LIN {X 0,Y 680.461,Z 406.458,A -85,B 0,C 180,E1 25579.128,E2 25579.128} C_VEL
LIN {X 0,Y 680.451,Z 406.465,A -85,B 0,C 180,E1 25576.563,E2 25576.563} C_VEL
LIN {X 0,Y 680.527,Z 406.447,A -85,B 0,C 180,E1 25573.683,E2 25573.683} C_VEL
LIN {X 0,Y 680.452,Z 406.461,A -85,B 0,C 180,E1 25570.756,E2 25570.756} C_VEL
LIN {X 0,Y 680.448,Z 406.447,A -85,B 0,C 180,E1 25568.195,E2 25568.195} C_VEL
LIN {X 0,Y 680.527,Z 406.46,A -85,B 0,C 180,E1 25565.311,E2 25565.311} C_VEL
LIN {X 0,Y 680.442,Z 406.447,A -85,B 0,C 180,E1 25562.358,E2 25562.358} C_VEL
LIN {X 0,Y 680.451,Z 406.466,A -85,B 0,C 180,E1 25559.832,E2 25559.832} C_VEL
LIN {X 0,Y 680.505,Z 406.442,A -85,B 0,C 180,E1 25556.799,E2 25556.799} C_VEL
LIN {X 0,Y 680.44,Z 406.466,A -85,B 0,C 180,E1 25554.011,E2 25554.011} C_VEL
LIN {X 0,Y 680.446,Z 406.46,A -85,B 0,C 180,E1 25551.55,E2 25551.55} C_VEL
LIN {X 0,Y 680.503,Z 406.464,A -85,B 0,C 180,E1 25548.51,E2 25548.51} C_VEL
LIN {X 0,Y 680.436,Z 406.455,A -85,B 0,C 180,E1 25545.794,E2 25545.794} C_VEL
LIN {X 0,Y 680.437,Z 406.459,A -85,B 0,C 180,E1 25543.338,E2 25543.338} C_VEL
LIN {X 0,Y 680.522,Z 406.444,A -85,B 0,C 180,E1 25540.427,E2 25540.427} C_VEL
LIN {X 0,Y 680.436,Z 406.465,A -85,B 0,C 180,E1 25537.538,E2 25537.538} C_VEL
LIN {X 0,Y 680.434,Z 406.459,A -85,B 0,C 180,E1 25535.038,E2 25535.038} C_VEL
LIN {X 0,Y 680.519,Z 406.463,A -85,B 0,C 180,E1 25532.049,E2 25532.049} C_VEL
LIN {X 0,Y 680.431,Z 406.462,A -85,B 0,C 180,E1 25529.244,E2 25529.244} C_VEL
LIN {X 0,Y 680.43,Z 406.467,A -85,B 0,C 180,E1 25526.762,E2 25526.762} C_VEL
LIN {X 0,Y 680.516,Z 406.467,A -85,B 0,C 180,E1 25523.9,E2 25523.9} C_VEL
LIN {X 0,Y 680.432,Z 406.473,A -85,B 0,C 180,E1 25521.012,E2 25521.012} C_VEL
LIN {X 0,Y 680.426,Z 406.493,A -85,B 0,C 180,E1 25518.714,E2 25518.714} C_VEL
LIN {X 0,Y 681.564,Z 409.672,A -85,B 0,C 180,E1 25518.35,E2 25518.35} C_VEL
LIN {X 0,Y 682.745,Z 411.865,A -85,B 0,C 180,E1 25518.064,E2 25518.064} C_VEL
LIN {X 0,Y 690.51,Z 428.251,A -85,B 0,C 180,E1 25516.112,E2 25516.112} C_VEL
LIN {X 0,Y 698.322,Z 440.196,A -85,B 0,C 180,E1 25515.278,E2 25515.278} C_VEL
LIN {X 0,Y 700.79,Z 450.164,A -85,B 0,C 180,E1 25514.933,E2 25514.933} C_VEL
LIN {X 0,Y 698.561,Z 650.685,A -85,B 0,C 180,E1 25512.321,E2 25512.321} C_VEL
LIN {X 0,Y 696.219,Z 875.891,A -85,B 0,C 180,E1 25509.482,E2 25509.482} C_VEL
LIN {X 0,Y 695.65,Z 912.99,A -85,B 0,C 180,E1 25508.982,E2 25508.982} C_VEL
LIN {X 0,Y 694.867,Z 939.914,A -85,B 0,C 180,E1 25508.45,E2 25508.45} C_VEL
LIN {X 0,Y 694.006,Z 964.483,A -85,B 0,C 180,E1 25507.821,E2 25507.821} C_VEL
LIN {X 0,Y 692.884,Z 992.482,A -85,B 0,C 180,E1 25506.92,E2 25506.92} C_VEL
LIN {X 0,Y 691.785,Z 1015.446,A -85,B 0,C 180,E1 25506.029,E2 25506.029} C_VEL
LIN {X 0,Y 690.755,Z 1035.669,A -85,B 0,C 180,E1 25505.129,E2 25505.129} C_VEL
LIN {X 0,Y 689.672,Z 1055.672,A -85,B 0,C 180,E1 25504.122,E2 25504.122} C_VEL
LIN {X 0,Y 688.5,Z 1076.88,A -85,B 0,C 180,E1 25502.921,E2 25502.921} C_VEL
LIN {X 0,Y 687.043,Z 1101.699,A -85,B 0,C 180,E1 25501.318,E2 25501.318} C_VEL
LIN {X 0,Y 685.98,Z 1120.495,A -85,B 0,C 180,E1 25499.945,E2 25499.945} C_VEL
LIN {X 0,Y 684.979,Z 1138.865,A -85,B 0,C 180,E1 25498.46,E2 25498.46} C_VEL
LIN {X 0,Y 683.778,Z 1160.458,A -85,B 0,C 180,E1 25496.5,E2 25496.5} C_VEL
LIN {X 0,Y 682.976,Z 1176.724,A -85,B 0,C 180,E1 25494.842,E2 25494.842} C_VEL
LIN {X 0,Y 682.182,Z 1193.517,A -85,B 0,C 180,E1 25492.943,E2 25492.943} C_VEL
LIN {X 0,Y 681.485,Z 1209.919,A -85,B 0,C 180,E1 25490.832,E2 25490.832} C_VEL
LIN {X 0,Y 681.039,Z 1222.568,A -85,B 0,C 180,E1 25489.001,E2 25489.001} C_VEL
LIN {X 0,Y 680.648,Z 1234.89,A -85,B 0,C 180,E1 25486.993,E2 25486.993} C_VEL
LIN {X 0,Y 680.344,Z 1246.853,A -85,B 0,C 180,E1 25484.726,E2 25484.726} C_VEL
LIN {X 0,Y 680.165,Z 1255.449,A -85,B 0,C 180,E1 25482.822,E2 25482.822} C_VEL
LIN {X 0,Y 680.027,Z 1262.449,A -85,B 0,C 180,E1 25481.017,E2 25481.017} C_VEL
LIN {X 0,Y 679.932,Z 1268.06,A -85,B 0,C 180,E1 25479.306,E2 25479.306} C_VEL
LIN {X 0,Y 679.922,Z 1273.174,A -85,B 0,C 180,E1 25477.433,E2 25477.433} C_VEL
LIN {X 0,Y 679.916,Z 1277.787,A -85,B 0,C 180,E1 25475.144,E2 25475.144} C_VEL
LIN {X 0,Y 679.912,Z 1280.543,A -85,B 0,C 180,E1 25472.948,E2 25472.948} C_VEL
LIN {X 0,Y 679.88,Z 1281.715,A -85,B 0,C 180,E1 25471.093,E2 25471.093} C_VEL
LIN {X 0,Y 679.863,Z 1281.826,A -85,B 0,C 180,E1 25469.323,E2 25469.323} C_VEL
LIN {X 0,Y 679.906,Z 1280.944,A -85,B 0,C 180,E1 25467.553,E2 25467.553} C_VEL
LIN {X 0,Y 679.915,Z 1278.916,A -85,B 0,C 180,E1 25465.612,E2 25465.612} C_VEL
LIN {X 0,Y 679.929,Z 1274.902,A -85,B 0,C 180,E1 25463.326,E2 25463.326} C_VEL
LIN {X 0,Y 679.942,Z 1269.325,A -85,B 0,C 180,E1 25461.116,E2 25461.116} C_VEL
LIN {X 0,Y 680.018,Z 1263.349,A -85,B 0,C 180,E1 25459.236,E2 25459.236} C_VEL
LIN {X 0,Y 680.138,Z 1256.5,A -85,B 0,C 180,E1 25457.431,E2 25457.431} C_VEL
LIN {X 0,Y 680.313,Z 1248.061,A -85,B 0,C 180,E1 25455.529,E2 25455.529} C_VEL
LIN {X 0,Y 680.558,Z 1237.337,A -85,B 0,C 180,E1 25453.438,E2 25453.438} C_VEL
LIN {X 0,Y 681.006,Z 1223.582,A -85,B 0,C 180,E1 25451.153,E2 25451.153} C_VEL
LIN {X 0,Y 681.419,Z 1211.446,A -85,B 0,C 180,E1 25449.379,E2 25449.379} C_VEL
LIN {X 0,Y 681.994,Z 1197.829,A -85,B 0,C 180,E1 25447.591,E2 25447.591} C_VEL
LIN {X 0,Y 682.821,Z 1180.065,A -85,B 0,C 180,E1 25445.516,E2 25445.516} C_VEL
LIN {X 0,Y 683.651,Z 1163.367,A -85,B 0,C 180,E1 25443.786,E2 25443.786} C_VEL
LIN {X 0,Y 684.531,Z 1146.227,A -85,B 0,C 180,E1 25442.179,E2 25442.179} C_VEL
LIN {X 0,Y 685.783,Z 1124.207,A -85,B 0,C 180,E1 25440.341,E2 25440.341} C_VEL
LIN {X 0,Y 686.866,Z 1105.212,A -85,B 0,C 180,E1 25438.931,E2 25438.931} C_VEL
LIN {X 0,Y 687.971,Z 1085.491,A -85,B 0,C 180,E1 25437.61,E2 25437.61} C_VEL
LIN {X 0,Y 689.442,Z 1059.964,A -85,B 0,C 180,E1 25436.107,E2 25436.107} C_VEL
LIN {X 0,Y 690.596,Z 1038.67,A -85,B 0,C 180,E1 25435.015,E2 25435.015} C_VEL
LIN {X 0,Y 691.623,Z 1018.703,A -85,B 0,C 180,E1 25434.109,E2 25434.109} C_VEL
LIN {X 0,Y 692.595,Z 998.275,A -85,B 0,C 180,E1 25433.295,E2 25433.295} C_VEL
LIN {X 0,Y 693.53,Z 975.906,A -85,B 0,C 180,E1 25432.524,E2 25432.524} C_VEL
LIN {X 0,Y 694.564,Z 949.817,A -85,B 0,C 180,E1 25431.784,E2 25431.784} C_VEL
LIN {X 0,Y 695.356,Z 923.501,A -85,B 0,C 180,E1 25431.208,E2 25431.208} C_VEL
LIN {X 0,Y 695.924,Z 898.793,A -85,B 0,C 180,E1 25430.808,E2 25430.808} C_VEL
LIN {X 0,Y 698.307,Z 673.627,A -85,B 0,C 180,E1 25427.971,E2 25427.971} C_VEL
LIN {X 0,Y 700.497,Z 475.392,A -85,B 0,C 180,E1 25425.4,E2 25425.4} C_VEL
LIN {X 0,Y 700.649,Z 448.932,A -85,B 0,C 180,E1 25425.038,E2 25425.038} C_VEL
LIN {X 0,Y 697.841,Z 439.159,A -85,B 0,C 180,E1 25424.667,E2 25424.667} C_VEL
LIN {X 0,Y 690.054,Z 427.342,A -85,B 0,C 180,E1 25423.812,E2 25423.812} C_VEL
LIN {X 0,Y 683.62,Z 413.795,A -85,B 0,C 180,E1 25422.172,E2 25422.172} C_VEL
LIN {X 0,Y 681.91,Z 410.194,A -85,B 0,C 180,E1 25421.724,E2 25421.724} C_VEL
LIN {X 0,Y 680.512,Z 407.036,A -85,B 0,C 180,E1 25421.338,E2 25421.338} C_VEL
LIN {X 0,Y 680.421,Z 406.454,A -85,B 0,C 180,E1 25421.258,E2 25421.258} C_VEL
LIN {X 0,Y 680.51,Z 406.449,A -85,B 0,C 180,E1 25418.428,E2 25418.428} C_VEL
LIN {X 0,Y 680.436,Z 406.469,A -85,B 0,C 180,E1 25415.482,E2 25415.482} C_VEL
LIN {X 0,Y 680.436,Z 406.462,A -85,B 0,C 180,E1 25413.037,E2 25413.037} C_VEL
LIN {X 0,Y 680.529,Z 406.444,A -85,B 0,C 180,E1 25410.165,E2 25410.165} C_VEL
LIN {X 0,Y 680.45,Z 406.466,A -85,B 0,C 180,E1 25407.25,E2 25407.25} C_VEL
LIN {X 0,Y 680.457,Z 406.449,A -85,B 0,C 180,E1 25404.666,E2 25404.666} C_VEL
LIN {X 0,Y 680.512,Z 406.452,A -85,B 0,C 180,E1 25401.642,E2 25401.642} C_VEL
LIN {X 0,Y 680.456,Z 406.459,A -85,B 0,C 180,E1 25398.859,E2 25398.859} C_VEL
LIN {X 0,Y 680.513,Z 406.451,A -85,B 0,C 180,E1 25396.036,E2 25396.036} C_VEL
LIN {X 0,Y 680.476,Z 406.46,A -85,B 0,C 180,E1 25392.992,E2 25392.992} C_VEL
LIN {X 0,Y 680.483,Z 406.459,A -85,B 0,C 180,E1 25390.241,E2 25390.241} C_VEL
LIN {X 0,Y 680.508,Z 406.458,A -85,B 0,C 180,E1 25387.09,E2 25387.09} C_VEL
LIN {X 0,Y 680.483,Z 406.459,A -85,B 0,C 180,E1 25384.213,E2 25384.213} C_VEL
LIN {X 0,Y 680.525,Z 406.457,A -85,B 0,C 180,E1 25381.179,E2 25381.179} C_VEL
LIN {X 0,Y 680.485,Z 406.459,A -85,B 0,C 180,E1 25378.232,E2 25378.232} C_VEL
LIN {X 0,Y 680.518,Z 406.46,A -85,B 0,C 180,E1 25375.28,E2 25375.28} C_VEL
LIN {X 0,Y 680.494,Z 406.456,A -85,B 0,C 180,E1 25372.316,E2 25372.316} C_VEL
LIN {X 0,Y 680.517,Z 406.456,A -85,B 0,C 180,E1 25369.331,E2 25369.331} C_VEL
LIN {X 0,Y 680.509,Z 406.452,A -85,B 0,C 180,E1 25366.316,E2 25366.316} C_VEL
LIN {X 0,Y 680.519,Z 406.46,A -85,B 0,C 180,E1 25363.263,E2 25363.263} C_VEL
LIN {X 0,Y 680.515,Z 406.446,A -85,B 0,C 180,E1 25360.159,E2 25360.159} C_VEL
LIN {X 0,Y 680.513,Z 406.465,A -85,B 0,C 180,E1 25357.085,E2 25357.085} C_VEL
LIN {X 0,Y 680.52,Z 406.44,A -85,B 0,C 180,E1 25354.033,E2 25354.033} C_VEL
LIN {X 0,Y 680.509,Z 406.452,A -85,B 0,C 180,E1 25350.956,E2 25350.956} C_VEL
LIN {X 0,Y 680.514,Z 406.444,A -85,B 0,C 180,E1 25349.429,E2 25349.429} C_VEL
LIN {X 0,Y 679.535,Z 406.579,A -85,B 0,C 180,E1 25348.78,E2 25348.78} C_VEL
LIN {X 0,Y 673.085,Z 407.384,A -85,B 0,C 180,E1 25346.963,E2 25346.963} C_VEL
LIN {X 0,Y 672.552,Z 407.44,A -85,B 0,C 180,E1 25346.49,E2 25346.49} C_VEL
LIN {X 0,Y 672.581,Z 407.453,A -85,B 0,C 180,E1 25343.511,E2 25343.511} C_VEL
LIN {X 0,Y 672.548,Z 407.456,A -85,B 0,C 180,E1 25340.482,E2 25340.482} C_VEL
LIN {X 0,Y 672.577,Z 407.645,A -85,B 0,C 180,E1 25338.551,E2 25338.551} C_VEL
LIN {X 0,Y 673.992,Z 411.125,A -85,B 0,C 180,E1 25338.118,E2 25338.118} C_VEL
LIN {X 0,Y 677.306,Z 418.165,A -85,B 0,C 180,E1 25337.242,E2 25337.242} C_VEL
LIN {X 0,Y 690.16,Z 436.862,A -85,B 0,C 180,E1 25335.824,E2 25335.824} C_VEL
LIN {X 0,Y 695.097,Z 444.613,A -85,B 0,C 180,E1 25335.294,E2 25335.294} C_VEL
LIN {X 0,Y 692.495,Z 652.368,A -85,B 0,C 180,E1 25332.574,E2 25332.574} C_VEL
LIN {X 0,Y 689.915,Z 876.906,A -85,B 0,C 180,E1 25329.723,E2 25329.723} C_VEL
LIN {X 0,Y 689.283,Z 907.492,A -85,B 0,C 180,E1 25329.277,E2 25329.277} C_VEL
LIN {X 0,Y 688.468,Z 932.192,A -85,B 0,C 180,E1 25328.77,E2 25328.77} C_VEL
LIN {X 0,Y 687.491,Z 957.703,A -85,B 0,C 180,E1 25328.098,E2 25328.098} C_VEL
LIN {X 0,Y 686.246,Z 984.6,A -85,B 0,C 180,E1 25327.206,E2 25327.206} C_VEL
LIN {X 0,Y 685.151,Z 1005.466,A -85,B 0,C 180,E1 25326.388,E2 25326.388} C_VEL
LIN {X 0,Y 684.005,Z 1025.807,A -85,B 0,C 180,E1 25325.475,E2 25325.475} C_VEL
LIN {X 0,Y 682.824,Z 1045.645,A -85,B 0,C 180,E1 25324.469,E2 25324.469} C_VEL
LIN {X 0,Y 681.518,Z 1066.981,A -85,B 0,C 180,E1 25323.251,E2 25323.251} C_VEL
LIN {X 0,Y 679.929,Z 1091.276,A -85,B 0,C 180,E1 25321.669,E2 25321.669} C_VEL
LIN {X 0,Y 678.72,Z 1110.473,A -85,B 0,C 180,E1 25320.255,E2 25320.255} C_VEL
LIN {X 0,Y 677.602,Z 1128.839,A -85,B 0,C 180,E1 25318.756,E2 25318.756} C_VEL
LIN {X 0,Y 676.295,Z 1150.13,A -85,B 0,C 180,E1 25316.805,E2 25316.805} C_VEL
LIN {X 0,Y 675.369,Z 1166.266,A -85,B 0,C 180,E1 25315.146,E2 25315.146} C_VEL
LIN {X 0,Y 674.542,Z 1182.325,A -85,B 0,C 180,E1 25313.316,E2 25313.316} C_VEL
LIN {X 0,Y 673.736,Z 1199.196,A -85,B 0,C 180,E1 25311.141,E2 25311.141} C_VEL
LIN {X 0,Y 673.208,Z 1212.129,A -85,B 0,C 180,E1 25309.254,E2 25309.254} C_VEL
LIN {X 0,Y 672.776,Z 1223.563,A -85,B 0,C 180,E1 25307.383,E2 25307.383} C_VEL
LIN {X 0,Y 672.406,Z 1236.211,A -85,B 0,C 180,E1 25304.997,E2 25304.997} C_VEL
LIN {X 0,Y 672.191,Z 1245.602,A -85,B 0,C 180,E1 25302.895,E2 25302.895} C_VEL
LIN {X 0,Y 672.049,Z 1252.579,A -85,B 0,C 180,E1 25301.067,E2 25301.067} C_VEL
LIN {X 0,Y 671.94,Z 1258.169,A -85,B 0,C 180,E1 25299.337,E2 25299.337} C_VEL
LIN {X 0,Y 671.92,Z 1263.258,A -85,B 0,C 180,E1 25297.441,E2 25297.441} C_VEL
LIN {X 0,Y 671.916,Z 1267.7,A -85,B 0,C 180,E1 25295.21,E2 25295.21} C_VEL
LIN {X 0,Y 671.911,Z 1270.503,A -85,B 0,C 180,E1 25292.988,E2 25292.988} C_VEL
LIN {X 0,Y 671.88,Z 1271.725,A -85,B 0,C 180,E1 25291.026,E2 25291.026} C_VEL
LIN {X 0,Y 671.863,Z 1271.817,A -85,B 0,C 180,E1 25289.235,E2 25289.235} C_VEL
LIN {X 0,Y 671.904,Z 1270.917,A -85,B 0,C 180,E1 25287.444,E2 25287.444} C_VEL
LIN {X 0,Y 671.911,Z 1268.866,A -85,B 0,C 180,E1 25285.479,E2 25285.479} C_VEL
LIN {X 0,Y 671.928,Z 1264.831,A -85,B 0,C 180,E1 25283.166,E2 25283.166} C_VEL
LIN {X 0,Y 671.944,Z 1259.472,A -85,B 0,C 180,E1 25281.014,E2 25281.014} C_VEL
LIN {X 0,Y 672.028,Z 1253.526,A -85,B 0,C 180,E1 25279.111,E2 25279.111} C_VEL
LIN {X 0,Y 672.179,Z 1246.349,A -85,B 0,C 180,E1 25277.198,E2 25277.198} C_VEL
LIN {X 0,Y 672.363,Z 1238.295,A -85,B 0,C 180,E1 25275.359,E2 25275.359} C_VEL
LIN {X 0,Y 672.626,Z 1228.064,A -85,B 0,C 180,E1 25273.331,E2 25273.331} C_VEL
LIN {X 0,Y 673.118,Z 1214.475,A -85,B 0,C 180,E1 25271.019,E2 25271.019} C_VEL
LIN {X 0,Y 673.606,Z 1201.803,A -85,B 0,C 180,E1 25269.134,E2 25269.134} C_VEL
LIN {X 0,Y 674.234,Z 1188.219,A -85,B 0,C 180,E1 25267.324,E2 25267.324} C_VEL
LIN {X 0,Y 675.186,Z 1170.313,A -85,B 0,C 180,E1 25265.204,E2 25265.204} C_VEL
LIN {X 0,Y 676.1,Z 1153.397,A -85,B 0,C 180,E1 25263.429,E2 25263.429} C_VEL
LIN {X 0,Y 677.123,Z 1136.253,A -85,B 0,C 180,E1 25261.805,E2 25261.805} C_VEL
LIN {X 0,Y 678.509,Z 1114.078,A -85,B 0,C 180,E1 25259.935,E2 25259.935} C_VEL
LIN {X 0,Y 679.729,Z 1094.572,A -85,B 0,C 180,E1 25258.475,E2 25258.475} C_VEL
LIN {X 0,Y 681.026,Z 1074.12,A -85,B 0,C 180,E1 25257.1,E2 25257.1} C_VEL
LIN {X 0,Y 682.626,Z 1049.079,A -85,B 0,C 180,E1 25255.626,E2 25255.626} C_VEL
LIN {X 0,Y 683.902,Z 1027.662,A -85,B 0,C 180,E1 25254.524,E2 25254.524} C_VEL
LIN {X 0,Y 685.039,Z 1007.552,A -85,B 0,C 180,E1 25253.611,E2 25253.611} C_VEL
LIN {X 0,Y 686.085,Z 987.66,A -85,B 0,C 180,E1 25252.818,E2 25252.818} C_VEL
LIN {X 0,Y 687.13,Z 965.185,A -85,B 0,C 180,E1 25252.043,E2 25252.043} C_VEL
LIN {X 0,Y 688.273,Z 938.268,A -85,B 0,C 180,E1 25251.284,E2 25251.284} C_VEL
LIN {X 0,Y 689.108,Z 912.632,A -85,B 0,C 180,E1 25250.727,E2 25250.727} C_VEL
LIN {X 0,Y 689.74,Z 887.818,A -85,B 0,C 180,E1 25250.328,E2 25250.328} C_VEL
LIN {X 0,Y 692.374,Z 662.26,A -85,B 0,C 180,E1 25247.464,E2 25247.464} C_VEL
LIN {X 0,Y 694.923,Z 457.036,A -85,B 0,C 180,E1 25244.78,E2 25244.78} C_VEL
LIN {X 0,Y 694.963,Z 444.111,A -85,B 0,C 180,E1 25244.597,E2 25244.597} C_VEL
LIN {X 0,Y 681.325,Z 423.894,A -85,B 0,C 180,E1 25243.12,E2 25243.12} C_VEL
LIN {X 0,Y 677.021,Z 417.66,A -85,B 0,C 180,E1 25242.622,E2 25242.622} C_VEL
LIN {X 0,Y 673.899,Z 411.027,A -85,B 0,C 180,E1 25241.775,E2 25241.775} C_VEL
LIN {X 0,Y 672.527,Z 407.436,A -85,B 0,C 180,E1 25241.31,E2 25241.31} C_VEL
LIN {X 0,Y 672.583,Z 407.454,A -85,B 0,C 180,E1 25238.292,E2 25238.292} C_VEL
LIN {X 0,Y 672.52,Z 407.454,A -85,B 0,C 180,E1 25235.44,E2 25235.44} C_VEL
LIN {X 0,Y 672.559,Z 407.45,A -85,B 0,C 180,E1 25232.661,E2 25232.661} C_VEL
LIN {X 0,Y 672.533,Z 407.44,A -85,B 0,C 180,E1 25229.578,E2 25229.578} C_VEL
LIN {X 0,Y 672.517,Z 407.454,A -85,B 0,C 180,E1 25226.967,E2 25226.967} C_VEL
LIN {X 0,Y 672.588,Z 407.442,A -85,B 0,C 180,E1 25224.038,E2 25224.038} C_VEL
LIN {X 0,Y 672.516,Z 407.442,A -85,B 0,C 180,E1 25221.088,E2 25221.088} C_VEL
LIN {X 0,Y 672.522,Z 407.449,A -85,B 0,C 180,E1 25218.463,E2 25218.463} C_VEL
LIN {X 0,Y 672.569,Z 407.427,A -85,B 0,C 180,E1 25215.433,E2 25215.433} C_VEL
LIN {X 0,Y 672.508,Z 407.452,A -85,B 0,C 180,E1 25212.625,E2 25212.625} C_VEL
LIN {X 0,Y 672.538,Z 407.443,A -85,B 0,C 180,E1 25209.931,E2 25209.931} C_VEL
LIN {X 0,Y 672.529,Z 407.452,A -85,B 0,C 180,E1 25206.831,E2 25206.831} C_VEL
LIN {X 0,Y 672.503,Z 407.449,A -85,B 0,C 180,E1 25204.263,E2 25204.263} C_VEL
LIN {X 0,Y 672.56,Z 407.438,A -85,B 0,C 180,E1 25201.448,E2 25201.448} C_VEL
LIN {X 0,Y 672.518,Z 407.447,A -85,B 0,C 180,E1 25198.466,E2 25198.466} C_VEL
LIN {X 0,Y 672.5,Z 407.438,A -85,B 0,C 180,E1 25195.907,E2 25195.907} C_VEL
LIN {X 0,Y 672.57,Z 407.454,A -85,B 0,C 180,E1 25193.084,E2 25193.084} C_VEL
LIN {X 0,Y 672.506,Z 407.44,A -85,B 0,C 180,E1 25190.068,E2 25190.068} C_VEL
LIN {X 0,Y 672.499,Z 407.456,A -85,B 0,C 180,E1 25187.55,E2 25187.55} C_VEL
LIN {X 0,Y 672.583,Z 407.429,A -85,B 0,C 180,E1 25184.655,E2 25184.655} C_VEL
LIN {X 0,Y 672.501,Z 407.453,A -85,B 0,C 180,E1 25181.716,E2 25181.716} C_VEL
LIN {X 0,Y 672.495,Z 407.432,A -85,B 0,C 180,E1 25179.185,E2 25179.185} C_VEL
LIN {X 0,Y 672.582,Z 407.446,A -85,B 0,C 180,E1 25176.241,E2 25176.241} C_VEL
LIN {X 0,Y 672.492,Z 407.452,A -85,B 0,C 180,E1 25173.317,E2 25173.317} C_VEL
LIN {X 0,Y 672.493,Z 407.454,A -85,B 0,C 180,E1 25170.909,E2 25170.909} C_VEL
LIN {X 0,Y 672.58,Z 407.454,A -85,B 0,C 180,E1 25168.045,E2 25168.045} C_VEL
LIN {X 0,Y 672.49,Z 407.45,A -85,B 0,C 180,E1 25165.079,E2 25165.079} C_VEL
LIN {X 0,Y 672.493,Z 407.459,A -85,B 0,C 180,E1 25162.551,E2 25162.551} C_VEL
LIN {X 0,Y 672.563,Z 407.436,A -85,B 0,C 180,E1 25159.561,E2 25159.561} C_VEL
LIN {X 0,Y 672.57,Z 407.709,A -85,B 0,C 180,E1 25159.371,E2 25159.371} C_VEL
LIN {X 0,Y 673.708,Z 410.787,A -85,B 0,C 180,E1 25159.004,E2 25159.004} C_VEL
LIN {X 0,Y 674.92,Z 413.31,A -85,B 0,C 180,E1 25158.68,E2 25158.68} C_VEL
LIN {X 0,Y 679.079,Z 421.931,A -85,B 0,C 180,E1 25157.595,E2 25157.595} C_VEL
LIN {X 0,Y 682.242,Z 428.302,A -85,B 0,C 180,E1 25156.838,E2 25156.838} C_VEL
LIN {X 0,Y 693.373,Z 445.15,A -85,B 0,C 180,E1 25155.621,E2 25155.621} C_VEL
LIN {X 0,Y 695.087,Z 452.546,A -85,B 0,C 180,E1 25155.37,E2 25155.37} C_VEL
LIN {X 0,Y 692.614,Z 652.848,A -85,B 0,C 180,E1 25152.741,E2 25152.741} C_VEL
LIN {X 0,Y 690.015,Z 878.054,A -85,B 0,C 180,E1 25149.879,E2 25149.879} C_VEL
LIN {X 0,Y 689.393,Z 913.685,A -85,B 0,C 180,E1 25149.39,E2 25149.39} C_VEL
LIN {X 0,Y 688.544,Z 940.238,A -85,B 0,C 180,E1 25148.86,E2 25148.86} C_VEL
LIN {X 0,Y 687.611,Z 964.53,A -85,B 0,C 180,E1 25148.234,E2 25148.234} C_VEL
LIN {X 0,Y 686.378,Z 992.125,A -85,B 0,C 180,E1 25147.344,E2 25147.344} C_VEL
LIN {X 0,Y 685.15,Z 1015.443,A -85,B 0,C 180,E1 25146.434,E2 25146.434} C_VEL
LIN {X 0,Y 684.005,Z 1035.795,A -85,B 0,C 180,E1 25145.521,E2 25145.521} C_VEL
LIN {X 0,Y 682.826,Z 1055.62,A -85,B 0,C 180,E1 25144.516,E2 25144.516} C_VEL
LIN {X 0,Y 681.499,Z 1077.329,A -85,B 0,C 180,E1 25143.275,E2 25143.275} C_VEL
LIN {X 0,Y 679.882,Z 1101.964,A -85,B 0,C 180,E1 25141.666,E2 25141.666} C_VEL
LIN {X 0,Y 678.728,Z 1120.322,A -85,B 0,C 180,E1 25140.312,E2 25140.312} C_VEL
LIN {X 0,Y 677.629,Z 1138.312,A -85,B 0,C 180,E1 25138.845,E2 25138.845} C_VEL
LIN {X 0,Y 676.291,Z 1160.16,A -85,B 0,C 180,E1 25136.847,E2 25136.847} C_VEL
LIN {X 0,Y 675.386,Z 1175.872,A -85,B 0,C 180,E1 25135.234,E2 25135.234} C_VEL
LIN {X 0,Y 674.604,Z 1191.204,A -85,B 0,C 180,E1 25133.494,E2 25133.494} C_VEL
LIN {X 0,Y 673.76,Z 1208.71,A -85,B 0,C 180,E1 25131.254,E2 25131.254} C_VEL
LIN {X 0,Y 673.218,Z 1221.869,A -85,B 0,C 180,E1 25129.339,E2 25129.339} C_VEL
LIN {X 0,Y 672.774,Z 1233.63,A -85,B 0,C 180,E1 25127.416,E2 25127.416} C_VEL
LIN {X 0,Y 672.399,Z 1246.444,A -85,B 0,C 180,E1 25124.992,E2 25124.992} C_VEL
LIN {X 0,Y 672.192,Z 1255.45,A -85,B 0,C 180,E1 25122.977,E2 25122.977} C_VEL
LIN {X 0,Y 672.05,Z 1262.45,A -85,B 0,C 180,E1 25121.149,E2 25121.149} C_VEL
LIN {X 0,Y 671.943,Z 1268.061,A -85,B 0,C 180,E1 25119.418,E2 25119.418} C_VEL
LIN {X 0,Y 671.923,Z 1273.171,A -85,B 0,C 180,E1 25117.522,E2 25117.522} C_VEL
LIN {X 0,Y 671.916,Z 1277.639,A -85,B 0,C 180,E1 25115.291,E2 25115.291} C_VEL
LIN {X 0,Y 671.91,Z 1280.475,A -85,B 0,C 180,E1 25113.068,E2 25113.068} C_VEL
LIN {X 0,Y 671.881,Z 1281.715,A -85,B 0,C 180,E1 25111.106,E2 25111.106} C_VEL
LIN {X 0,Y 671.863,Z 1281.826,A -85,B 0,C 180,E1 25109.315,E2 25109.315} C_VEL
LIN {X 0,Y 671.906,Z 1280.945,A -85,B 0,C 180,E1 25107.524,E2 25107.524} C_VEL
LIN {X 0,Y 671.913,Z 1278.913,A -85,B 0,C 180,E1 25105.56,E2 25105.56} C_VEL
LIN {X 0,Y 671.929,Z 1274.902,A -85,B 0,C 180,E1 25103.247,E2 25103.247} C_VEL
LIN {X 0,Y 671.947,Z 1269.579,A -85,B 0,C 180,E1 25101.095,E2 25101.095} C_VEL
LIN {X 0,Y 672.033,Z 1263.349,A -85,B 0,C 180,E1 25099.106,E2 25099.106} C_VEL
LIN {X 0,Y 672.176,Z 1256.501,A -85,B 0,C 180,E1 25097.28,E2 25097.28} C_VEL
LIN {X 0,Y 672.368,Z 1248.063,A -85,B 0,C 180,E1 25095.354,E2 25095.354} C_VEL
LIN {X 0,Y 672.673,Z 1236.873,A -85,B 0,C 180,E1 25093.149,E2 25093.149} C_VEL
LIN {X 0,Y 673.152,Z 1223.583,A -85,B 0,C 180,E1 25090.925,E2 25090.925} C_VEL
LIN {X 0,Y 673.655,Z 1210.803,A -85,B 0,C 180,E1 25089.039,E2 25089.039} C_VEL
LIN {X 0,Y 674.369,Z 1195.629,A -85,B 0,C 180,E1 25087.038,E2 25087.038} C_VEL
LIN {X 0,Y 675.304,Z 1177.848,A -85,B 0,C 180,E1 25084.98,E2 25084.98} C_VEL
LIN {X 0,Y 676.176,Z 1161.97,A -85,B 0,C 180,E1 25083.332,E2 25083.332} C_VEL
LIN {X 0,Y 677.398,Z 1142.666,A -85,B 0,C 180,E1 25081.524,E2 25081.524} C_VEL
LIN {X 0,Y 678.615,Z 1122.24,A -85,B 0,C 180,E1 25079.837,E2 25079.837} C_VEL
LIN {X 0,Y 679.764,Z 1103.887,A -85,B 0,C 180,E1 25078.471,E2 25078.471} C_VEL
LIN {X 0,Y 681.2,Z 1081.901,A -85,B 0,C 180,E1 25077.004,E2 25077.004} C_VEL
LIN {X 0,Y 682.727,Z 1057.297,A -85,B 0,C 180,E1 25075.575,E2 25075.575} C_VEL
LIN {X 0,Y 683.959,Z 1036.686,A -85,B 0,C 180,E1 25074.522,E2 25074.522} C_VEL
LIN {X 0,Y 685.099,Z 1016.445,A -85,B 0,C 180,E1 25073.609,E2 25073.609} C_VEL
LIN {X 0,Y 686.227,Z 994.996,A -85,B 0,C 180,E1 25072.764,E2 25072.764} C_VEL
LIN {X 0,Y 687.509,Z 967.115,A -85,B 0,C 180,E1 25071.839,E2 25071.839} C_VEL
LIN {X 0,Y 688.482,Z 941.865,A -85,B 0,C 180,E1 25071.177,E2 25071.177} C_VEL
LIN {X 0,Y 689.299,Z 916.908,A -85,B 0,C 180,E1 25070.667,E2 25070.667} C_VEL
LIN {X 0,Y 689.938,Z 884.658,A -85,B 0,C 180,E1 25070.203,E2 25070.203} C_VEL
LIN {X 0,Y 692.523,Z 660.013,A -85,B 0,C 180,E1 25067.351,E2 25067.351} C_VEL
LIN {X 0,Y 694.974,Z 461.158,A -85,B 0,C 180,E1 25064.745,E2 25064.745} C_VEL
LIN {X 0,Y 694.945,Z 451.203,A -85,B 0,C 180,E1 25064.599,E2 25064.599} C_VEL
LIN {X 0,Y 692.933,Z 444.186,A -85,B 0,C 180,E1 25064.328,E2 25064.328} C_VEL
LIN {X 0,Y 681.791,Z 427.694,A -85,B 0,C 180,E1 25063.112,E2 25063.112} C_VEL
LIN {X 0,Y 676.078,Z 415.52,A -85,B 0,C 180,E1 25061.61,E2 25061.61} C_VEL
LIN {X 0,Y 673.709,Z 410.783,A -85,B 0,C 180,E1 25060.996,E2 25060.996} C_VEL
LIN {X 0,Y 672.548,Z 407.436,A -85,B 0,C 180,E1 25060.596,E2 25060.596} C_VEL
LIN {X 0,Y 672.495,Z 407.442,A -85,B 0,C 180,E1 25057.581,E2 25057.581} C_VEL
LIN {X 0,Y 672.494,Z 407.456,A -85,B 0,C 180,E1 25055.128,E2 25055.128} C_VEL
LIN {X 0,Y 672.566,Z 407.452,A -85,B 0,C 180,E1 25052.358,E2 25052.358} C_VEL
LIN {X 0,Y 672.51,Z 407.444,A -85,B 0,C 180,E1 25049.383,E2 25049.383} C_VEL
LIN {X 0,Y 672.51,Z 407.457,A -85,B 0,C 180,E1 25046.864,E2 25046.864} C_VEL
LIN {X 0,Y 672.588,Z 407.446,A -85,B 0,C 180,E1 25043.851,E2 25043.851} C_VEL
LIN {X 0,Y 672.515,Z 407.443,A -85,B 0,C 180,E1 25040.981,E2 25040.981} C_VEL
LIN {X 0,Y 672.56,Z 407.451,A -85,B 0,C 180,E1 25038.192,E2 25038.192} C_VEL
LIN {X 0,Y 672.533,Z 407.429,A -85,B 0,C 180,E1 25035.081,E2 25035.081} C_VEL
LIN {X 0,Y 672.537,Z 407.453,A -85,B 0,C 180,E1 25032.362,E2 25032.362} C_VEL
LIN {X 0,Y 672.574,Z 407.424,A -85,B 0,C 180,E1 25029.239,E2 25029.239} C_VEL
LIN {X 0,Y 672.539,Z 407.452,A -85,B 0,C 180,E1 25026.316,E2 25026.316} C_VEL
LIN {X 0,Y 672.582,Z 407.424,A -85,B 0,C 180,E1 25023.324,E2 25023.324} C_VEL
LIN {X 0,Y 672.545,Z 407.45,A -85,B 0,C 180,E1 25020.341,E2 25020.341} C_VEL
LIN {X 0,Y 672.579,Z 407.427,A -85,B 0,C 180,E1 25017.444,E2 25017.444} C_VEL
LIN {X 0,Y 672.553,Z 407.448,A -85,B 0,C 180,E1 25014.369,E2 25014.369} C_VEL
LIN {X 0,Y 672.582,Z 407.429,A -85,B 0,C 180,E1 25011.45,E2 25011.45} C_VEL
LIN {X 0,Y 672.568,Z 407.447,A -85,B 0,C 180,E1 25008.335,E2 25008.335} C_VEL
LIN {X 0,Y 672.577,Z 407.429,A -85,B 0,C 180,E1 25005.273,E2 25005.273} C_VEL
LIN {X 0,Y 672.573,Z 407.448,A -85,B 0,C 180,E1 25002.166,E2 25002.166} C_VEL
LIN {X 0,Y 672.572,Z 407.434,A -85,B 0,C 180,E1 24999.096,E2 24999.096} C_VEL
LIN {X 0,Y 672.581,Z 407.445,A -85,B 0,C 180,E1 24996.055,E2 24996.055} C_VEL
LIN {X 0,Y 672.568,Z 407.45,A -85,B 0,C 180,E1 24992.938,E2 24992.938} C_VEL
LIN {X 0,Y 672.586,Z 407.428,A -85,B 0,C 180,E1 24989.908,E2 24989.908} C_VEL
LIN {X 0,Y 672.563,Z 407.444,A -85,B 0,C 180,E1 24986.825,E2 24986.825} C_VEL
LIN {X 0,Y 672.552,Z 407.44,A -85,B 0,C 180,E1 24986.49,E2 24986.49} C_VEL
LIN {X 0,Y 671.572,Z 407.559,A -85,B 0,C 180,E1 24985.834,E2 24985.834} C_VEL
LIN {X 0,Y 665.177,Z 408.374,A -85,B 0,C 180,E1 24983.995,E2 24983.995} C_VEL
LIN {X 0,Y 664.642,Z 408.442,A -85,B 0,C 180,E1 24983.517,E2 24983.517} C_VEL
LIN {X 0,Y 664.609,Z 408.443,A -85,B 0,C 180,E1 24980.476,E2 24980.476} C_VEL
LIN {X 0,Y 664.645,Z 408.443,A -85,B 0,C 180,E1 24979.273,E2 24979.273} C_VEL
LIN {X 0,Y 665.818,Z 411.714,A -85,B 0,C 180,E1 24978.87,E2 24978.87} C_VEL
LIN {X 0,Y 666.949,Z 414.048,A -85,B 0,C 180,E1 24978.556,E2 24978.556} C_VEL
LIN {X 0,Y 669.13,Z 418.392,A -85,B 0,C 180,E1 24978.004,E2 24978.004} C_VEL
LIN {X 0,Y 684.846,Z 441.054,A -85,B 0,C 180,E1 24976.222,E2 24976.222} C_VEL
LIN {X 0,Y 689.41,Z 448.321,A -85,B 0,C 180,E1 24975.72,E2 24975.72} C_VEL
LIN {X 0,Y 686.562,Z 655.4,A -85,B 0,C 180,E1 24972.988,E2 24972.988} C_VEL
LIN {X 0,Y 683.716,Z 880.638,A -85,B 0,C 180,E1 24970.107,E2 24970.107} C_VEL
LIN {X 0,Y 683.026,Z 908.798,A -85,B 0,C 180,E1 24969.68,E2 24969.68} C_VEL
LIN {X 0,Y 682.165,Z 932.85,A -85,B 0,C 180,E1 24969.18,E2 24969.18} C_VEL
LIN {X 0,Y 681.071,Z 958.778,A -85,B 0,C 180,E1 24968.488,E2 24968.488} C_VEL
LIN {X 0,Y 679.712,Z 985.319,A -85,B 0,C 180,E1 24967.596,E2 24967.596} C_VEL
LIN {X 0,Y 678.487,Z 1006.607,A -85,B 0,C 180,E1 24966.751,E2 24966.751} C_VEL
LIN {X 0,Y 677.219,Z 1027.124,A -85,B 0,C 180,E1 24965.818,E2 24965.818} C_VEL
LIN {X 0,Y 675.839,Z 1048.303,A -85,B 0,C 180,E1 24964.723,E2 24964.723} C_VEL
LIN {X 0,Y 674.166,Z 1072.717,A -85,B 0,C 180,E1 24963.283,E2 24963.283} C_VEL
LIN {X 0,Y 672.632,Z 1093.952,A -85,B 0,C 180,E1 24961.853,E2 24961.853} C_VEL
LIN {X 0,Y 671.319,Z 1113.05,A -85,B 0,C 180,E1 24960.414,E2 24960.414} C_VEL
LIN {X 0,Y 669.823,Z 1135.25,A -85,B 0,C 180,E1 24958.536,E2 24958.536} C_VEL
LIN {X 0,Y 668.616,Z 1152.932,A -85,B 0,C 180,E1 24956.85,E2 24956.85} C_VEL
LIN {X 0,Y 667.64,Z 1168.815,A -85,B 0,C 180,E1 24955.173,E2 24955.173} C_VEL
LIN {X 0,Y 666.595,Z 1186.78,A -85,B 0,C 180,E1 24953.049,E2 24953.049} C_VEL
LIN {X 0,Y 665.859,Z 1201.136,A -85,B 0,C 180,E1 24951.126,E2 24951.126} C_VEL
LIN {X 0,Y 665.292,Z 1213.872,A -85,B 0,C 180,E1 24949.218,E2 24949.218} C_VEL
LIN {X 0,Y 664.738,Z 1227.573,A -85,B 0,C 180,E1 24946.878,E2 24946.878} C_VEL
LIN {X 0,Y 664.428,Z 1237.857,A -85,B 0,C 180,E1 24944.825,E2 24944.825} C_VEL
LIN {X 0,Y 664.212,Z 1246.32,A -85,B 0,C 180,E1 24942.875,E2 24942.875} C_VEL
LIN {X 0,Y 664.052,Z 1253.499,A -85,B 0,C 180,E1 24940.939,E2 24940.939} C_VEL
LIN {X 0,Y 663.962,Z 1260.21,A -85,B 0,C 180,E1 24938.751,E2 24938.751} C_VEL
LIN {X 0,Y 663.935,Z 1265.672,A -85,B 0,C 180,E1 24936.401,E2 24936.401} C_VEL
LIN {X 0,Y 663.918,Z 1269.306,A -85,B 0,C 180,E1 24934.148,E2 24934.148} C_VEL
LIN {X 0,Y 663.907,Z 1271.517,A -85,B 0,C 180,E1 24931.728,E2 24931.728} C_VEL
LIN {X 0,Y 663.869,Z 1271.884,A -85,B 0,C 180,E1 24929.485,E2 24929.485} C_VEL
LIN {X 0,Y 663.905,Z 1271.051,A -85,B 0,C 180,E1 24927.586,E2 24927.586} C_VEL
LIN {X 0,Y 663.912,Z 1268.976,A -85,B 0,C 180,E1 24925.511,E2 24925.511} C_VEL
LIN {X 0,Y 663.93,Z 1265.001,A -85,B 0,C 180,E1 24923.17,E2 24923.17} C_VEL
LIN {X 0,Y 663.949,Z 1259.724,A -85,B 0,C 180,E1 24920.992,E2 24920.992} C_VEL
LIN {X 0,Y 664.046,Z 1253.525,A -85,B 0,C 180,E1 24918.978,E2 24918.978} C_VEL
LIN {X 0,Y 664.212,Z 1246.348,A -85,B 0,C 180,E1 24917.041,E2 24917.041} C_VEL
LIN {X 0,Y 664.418,Z 1238.294,A -85,B 0,C 180,E1 24915.18,E2 24915.18} C_VEL
LIN {X 0,Y 664.723,Z 1228.063,A -85,B 0,C 180,E1 24913.127,E2 24913.127} C_VEL
LIN {X 0,Y 665.27,Z 1214.469,A -85,B 0,C 180,E1 24910.786,E2 24910.786} C_VEL
LIN {X 0,Y 665.838,Z 1201.516,A -85,B 0,C 180,E1 24908.838,E2 24908.838} C_VEL
LIN {X 0,Y 666.551,Z 1187.506,A -85,B 0,C 180,E1 24906.954,E2 24906.954} C_VEL
LIN {X 0,Y 667.625,Z 1169.116,A -85,B 0,C 180,E1 24904.77,E2 24904.77} C_VEL
LIN {X 0,Y 668.629,Z 1152.68,A -85,B 0,C 180,E1 24903.035,E2 24903.035} C_VEL
LIN {X 0,Y 669.905,Z 1134.215,A -85,B 0,C 180,E1 24901.279,E2 24901.279} C_VEL
LIN {X 0,Y 671.33,Z 1112.861,A -85,B 0,C 180,E1 24899.481,E2 24899.481} C_VEL
LIN {X 0,Y 672.637,Z 1093.896,A -85,B 0,C 180,E1 24898.053,E2 24898.053} C_VEL
LIN {X 0,Y 674.236,Z 1071.904,A -85,B 0,C 180,E1 24896.574,E2 24896.574} C_VEL
LIN {X 0,Y 675.901,Z 1047.29,A -85,B 0,C 180,E1 24895.131,E2 24895.131} C_VEL
LIN {X 0,Y 677.246,Z 1026.656,A -85,B 0,C 180,E1 24894.07,E2 24894.07} C_VEL
LIN {X 0,Y 678.496,Z 1006.404,A -85,B 0,C 180,E1 24893.15,E2 24893.15} C_VEL
LIN {X 0,Y 679.762,Z 984.364,A -85,B 0,C 180,E1 24892.277,E2 24892.277} C_VEL
LIN {X 0,Y 681.18,Z 956.227,A -85,B 0,C 180,E1 24891.347,E2 24891.347} C_VEL
LIN {X 0,Y 682.221,Z 931.44,A -85,B 0,C 180,E1 24890.698,E2 24890.698} C_VEL
LIN {X 0,Y 683.113,Z 906.238,A -85,B 0,C 180,E1 24890.182,E2 24890.182} C_VEL
LIN {X 0,Y 683.815,Z 872.537,A -85,B 0,C 180,E1 24889.701,E2 24889.701} C_VEL
LIN {X 0,Y 686.636,Z 649.802,A -85,B 0,C 180,E1 24886.849,E2 24886.849} C_VEL
LIN {X 0,Y 689.416,Z 448.009,A -85,B 0,C 180,E1 24884.186,E2 24884.186} C_VEL
LIN {X 0,Y 676.595,Z 429.109,A -85,B 0,C 180,E1 24882.771,E2 24882.771} C_VEL
LIN {X 0,Y 668.725,Z 417.542,A -85,B 0,C 180,E1 24881.826,E2 24881.826} C_VEL
LIN {X 0,Y 664.777,Z 409.163,A -85,B 0,C 180,E1 24880.713,E2 24880.713} C_VEL
LIN {X 0,Y 664.651,Z 408.424,A -85,B 0,C 180,E1 24880.591,E2 24880.591} C_VEL
LIN {X 0,Y 664.585,Z 408.446,A -85,B 0,C 180,E1 24877.651,E2 24877.651} C_VEL
LIN {X 0,Y 664.598,Z 408.428,A -85,B 0,C 180,E1 24874.928,E2 24874.928} C_VEL
LIN {X 0,Y 664.598,Z 408.439,A -85,B 0,C 180,E1 24871.673,E2 24871.673} C_VEL
LIN {X 0,Y 664.58,Z 408.433,A -85,B 0,C 180,E1 24868.977,E2 24868.977} C_VEL
LIN {X 0,Y 664.647,Z 408.417,A -85,B 0,C 180,E1 24866.058,E2 24866.058} C_VEL
LIN {X 0,Y 664.578,Z 408.443,A -85,B 0,C 180,E1 24863.122,E2 24863.122} C_VEL
LIN {X 0,Y 664.584,Z 408.425,A -85,B 0,C 180,E1 24860.521,E2 24860.521} C_VEL
LIN {X 0,Y 664.62,Z 408.44,A -85,B 0,C 180,E1 24857.421,E2 24857.421} C_VEL
LIN {X 0,Y 664.568,Z 408.417,A -85,B 0,C 180,E1 24854.641,E2 24854.641} C_VEL
LIN {X 0,Y 664.616,Z 408.444,A -85,B 0,C 180,E1 24851.895,E2 24851.895} C_VEL
LIN {X 0,Y 664.581,Z 408.417,A -85,B 0,C 180,E1 24848.828,E2 24848.828} C_VEL
LIN {X 0,Y 664.568,Z 408.444,A -85,B 0,C 180,E1 24846.219,E2 24846.219} C_VEL
LIN {X 0,Y 664.644,Z 408.414,A -85,B 0,C 180,E1 24843.277,E2 24843.277} C_VEL
LIN {X 0,Y 664.571,Z 408.443,A -85,B 0,C 180,E1 24840.345,E2 24840.345} C_VEL
LIN {X 0,Y 664.574,Z 408.436,A -85,B 0,C 180,E1 24837.758,E2 24837.758} C_VEL
LIN {X 0,Y 664.615,Z 408.442,A -85,B 0,C 180,E1 24834.648,E2 24834.648} C_VEL
LIN {X 0,Y 664.56,Z 408.435,A -85,B 0,C 180,E1 24831.956,E2 24831.956} C_VEL
LIN {X 0,Y 664.577,Z 408.43,A -85,B 0,C 180,E1 24829.335,E2 24829.335} C_VEL
LIN {X 0,Y 664.586,Z 408.43,A -85,B 0,C 180,E1 24826.159,E2 24826.159} C_VEL
LIN {X 0,Y 664.556,Z 408.435,A -85,B 0,C 180,E1 24823.569,E2 24823.569} C_VEL
LIN {X 0,Y 664.586,Z 408.441,A -85,B 0,C 180,E1 24820.944,E2 24820.944} C_VEL
LIN {X 0,Y 664.577,Z 408.443,A -85,B 0,C 180,E1 24817.812,E2 24817.812} C_VEL
LIN {X 0,Y 664.552,Z 408.435,A -85,B 0,C 180,E1 24815.274,E2 24815.274} C_VEL
LIN {X 0,Y 664.588,Z 408.443,A -85,B 0,C 180,E1 24812.571,E2 24812.571} C_VEL
LIN {X 0,Y 664.564,Z 408.431,A -85,B 0,C 180,E1 24809.433,E2 24809.433} C_VEL
LIN {X 0,Y 664.549,Z 408.446,A -85,B 0,C 180,E1 24806.895,E2 24806.895} C_VEL
LIN {X 0,Y 664.599,Z 408.445,A -85,B 0,C 180,E1 24804.178,E2 24804.178} C_VEL
LIN {X 0,Y 664.564,Z 408.451,A -85,B 0,C 180,E1 24801.14,E2 24801.14} C_VEL
LIN {X 0,Y 664.617,Z 408.648,A -85,B 0,C 180,E1 24800.085,E2 24800.085} C_VEL
LIN {X 0,Y 665.942,Z 411.901,A -85,B 0,C 180,E1 24799.674,E2 24799.674} C_VEL
LIN {X 0,Y 666.914,Z 413.926,A -85,B 0,C 180,E1 24799.406,E2 24799.406} C_VEL
LIN {X 0,Y 673.455,Z 427.729,A -85,B 0,C 180,E1 24797.649,E2 24797.649} C_VEL
LIN {X 0,Y 686.072,Z 446.115,A -85,B 0,C 180,E1 24796.233,E2 24796.233} C_VEL
LIN {X 0,Y 688.449,Z 450.21,A -85,B 0,C 180,E1 24795.966,E2 24795.966} C_VEL
LIN {X 0,Y 689.427,Z 454.743,A -85,B 0,C 180,E1 24795.816,E2 24795.816} C_VEL
LIN {X 0,Y 686.707,Z 654.706,A -85,B 0,C 180,E1 24793.172,E2 24793.172} C_VEL
LIN {X 0,Y 683.85,Z 879.836,A -85,B 0,C 180,E1 24790.288,E2 24790.288} C_VEL
LIN {X 0,Y 683.164,Z 914.599,A -85,B 0,C 180,E1 24789.802,E2 24789.802} C_VEL
LIN {X 0,Y 682.26,Z 940.478,A -85,B 0,C 180,E1 24789.28,E2 24789.28} C_VEL
LIN {X 0,Y 681.259,Z 964.403,A -85,B 0,C 180,E1 24788.659,E2 24788.659} C_VEL
LIN {X 0,Y 679.895,Z 991.994,A -85,B 0,C 180,E1 24787.767,E2 24787.767} C_VEL
LIN {X 0,Y 678.55,Z 1015.439,A -85,B 0,C 180,E1 24786.846,E2 24786.846} C_VEL
LIN {X 0,Y 677.296,Z 1035.79,A -85,B 0,C 180,E1 24785.927,E2 24785.927} C_VEL
LIN {X 0,Y 675.95,Z 1056.514,A -85,B 0,C 180,E1 24784.866,E2 24784.866} C_VEL
LIN {X 0,Y 674.354,Z 1080.518,A -85,B 0,C 180,E1 24783.471,E2 24783.471} C_VEL
LIN {X 0,Y 672.68,Z 1103.297,A -85,B 0,C 180,E1 24781.945,E2 24781.945} C_VEL
LIN {X 0,Y 671.429,Z 1121.285,A -85,B 0,C 180,E1 24780.598,E2 24780.598} C_VEL
LIN {X 0,Y 670.087,Z 1141.634,A -85,B 0,C 180,E1 24778.908,E2 24778.908} C_VEL
LIN {X 0,Y 668.709,Z 1161.558,A -85,B 0,C 180,E1 24777.032,E2 24777.032} C_VEL
LIN {X 0,Y 667.699,Z 1177.574,A -85,B 0,C 180,E1 24775.355,E2 24775.355} C_VEL
LIN {X 0,Y 666.712,Z 1195.032,A -85,B 0,C 180,E1 24773.32,E2 24773.32} C_VEL
LIN {X 0,Y 665.872,Z 1210.842,A -85,B 0,C 180,E1 24771.213,E2 24771.213} C_VEL
LIN {X 0,Y 665.303,Z 1223.671,A -85,B 0,C 180,E1 24769.295,E2 24769.295} C_VEL
LIN {X 0,Y 664.754,Z 1237.365,A -85,B 0,C 180,E1 24766.963,E2 24766.963} C_VEL
LIN {X 0,Y 664.422,Z 1248.087,A -85,B 0,C 180,E1 24764.82,E2 24764.82} C_VEL
LIN {X 0,Y 664.209,Z 1256.524,A -85,B 0,C 180,E1 24762.87,E2 24762.87} C_VEL
LIN {X 0,Y 664.047,Z 1263.673,A -85,B 0,C 180,E1 24760.934,E2 24760.934} C_VEL
LIN {X 0,Y 663.977,Z 1270.822,A -85,B 0,C 180,E1 24758.571,E2 24758.571} C_VEL
LIN {X 0,Y 663.933,Z 1276.098,A -85,B 0,C 180,E1 24756.222,E2 24756.222} C_VEL
LIN {X 0,Y 663.916,Z 1279.485,A -85,B 0,C 180,E1 24754.056,E2 24754.056} C_VEL
LIN {X 0,Y 663.91,Z 1281.602,A -85,B 0,C 180,E1 24751.551,E2 24751.551} C_VEL
LIN {X 0,Y 663.866,Z 1281.871,A -85,B 0,C 180,E1 24749.48,E2 24749.48} C_VEL
LIN {X 0,Y 663.907,Z 1281.012,A -85,B 0,C 180,E1 24747.581,E2 24747.581} C_VEL
LIN {X 0,Y 663.914,Z 1278.994,A -85,B 0,C 180,E1 24745.57,E2 24745.57} C_VEL
LIN {X 0,Y 663.931,Z 1275.074,A -85,B 0,C 180,E1 24743.252,E2 24743.252} C_VEL
LIN {X 0,Y 663.947,Z 1269.578,A -85,B 0,C 180,E1 24740.987,E2 24740.987} C_VEL
LIN {X 0,Y 664.051,Z 1263.35,A -85,B 0,C 180,E1 24738.973,E2 24738.973} C_VEL
LIN {X 0,Y 664.21,Z 1256.502,A -85,B 0,C 180,E1 24737.125,E2 24737.125} C_VEL
LIN {X 0,Y 664.422,Z 1248.064,A -85,B 0,C 180,E1 24735.175,E2 24735.175} C_VEL
LIN {X 0,Y 664.782,Z 1236.875,A -85,B 0,C 180,E1 24732.943,E2 24732.943} C_VEL
LIN {X 0,Y 665.307,Z 1223.582,A -85,B 0,C 180,E1 24730.691,E2 24730.691} C_VEL
LIN {X 0,Y 665.875,Z 1210.805,A -85,B 0,C 180,E1 24728.782,E2 24728.782} C_VEL
LIN {X 0,Y 666.717,Z 1194.99,A -85,B 0,C 180,E1 24726.675,E2 24726.675} C_VEL
LIN {X 0,Y 667.7,Z 1177.526,A -85,B 0,C 180,E1 24724.64,E2 24724.64} C_VEL
LIN {X 0,Y 668.714,Z 1161.505,A -85,B 0,C 180,E1 24722.962,E2 24722.962} C_VEL
LIN {X 0,Y 670.091,Z 1141.57,A -85,B 0,C 180,E1 24721.087,E2 24721.087} C_VEL
LIN {X 0,Y 671.43,Z 1121.282,A -85,B 0,C 180,E1 24719.402,E2 24719.402} C_VEL
LIN {X 0,Y 672.737,Z 1102.548,A -85,B 0,C 180,E1 24718.002,E2 24718.002} C_VEL
LIN {X 0,Y 674.462,Z 1078.808,A -85,B 0,C 180,E1 24716.426,E2 24716.426} C_VEL
LIN {X 0,Y 675.957,Z 1056.409,A -85,B 0,C 180,E1 24715.129,E2 24715.129} C_VEL
LIN {X 0,Y 677.304,Z 1035.677,A -85,B 0,C 180,E1 24714.067,E2 24714.067} C_VEL
LIN {X 0,Y 678.615,Z 1014.294,A -85,B 0,C 180,E1 24713.104,E2 24713.104} C_VEL
LIN {X 0,Y 680.142,Z 986.878,A -85,B 0,C 180,E1 24712.053,E2 24712.053} C_VEL
LIN {X 0,Y 681.354,Z 962.192,A -85,B 0,C 180,E1 24711.279,E2 24711.279} C_VEL
LIN {X 0,Y 682.354,Z 938.196,A -85,B 0,C 180,E1 24710.667,E2 24710.667} C_VEL
LIN {X 0,Y 683.28,Z 910.534,A -85,B 0,C 180,E1 24710.129,E2 24710.129} C_VEL
LIN {X 0,Y 684.044,Z 863.558,A -85,B 0,C 180,E1 24709.506,E2 24709.506} C_VEL
LIN {X 0,Y 686.895,Z 640.928,A -85,B 0,C 180,E1 24706.649,E2 24706.649} C_VEL
LIN {X 0,Y 689.438,Z 454.03,A -85,B 0,C 180,E1 24704.174,E2 24704.174} C_VEL
LIN {X 0,Y 687.977,Z 449.054,A -85,B 0,C 180,E1 24703.976,E2 24703.976} C_VEL
LIN {X 0,Y 677.358,Z 433.35,A -85,B 0,C 180,E1 24702.797,E2 24702.797} C_VEL
LIN {X 0,Y 673.2,Z 427.178,A -85,B 0,C 180,E1 24702.286,E2 24702.286} C_VEL
LIN {X 0,Y 667.863,Z 416.027,A -85,B 0,C 180,E1 24700.863,E2 24700.863} C_VEL
LIN {X 0,Y 665.938,Z 411.908,A -85,B 0,C 180,E1 24700.326,E2 24700.326} C_VEL
LIN {X 0,Y 664.571,Z 408.445,A -85,B 0,C 180,E1 24699.863,E2 24699.863} C_VEL
LIN {X 0,Y 664.549,Z 408.433,A -85,B 0,C 180,E1 24697.255,E2 24697.255} C_VEL
LIN {X 0,Y 664.613,Z 408.424,A -85,B 0,C 180,E1 24694.467,E2 24694.467} C_VEL
LIN {X 0,Y 664.571,Z 408.444,A -85,B 0,C 180,E1 24691.451,E2 24691.451} C_VEL
LIN {X 0,Y 664.569,Z 408.435,A -85,B 0,C 180,E1 24688.877,E2 24688.877} C_VEL
LIN {X 0,Y 664.645,Z 408.418,A -85,B 0,C 180,E1 24685.962,E2 24685.962} C_VEL
LIN {X 0,Y 664.574,Z 408.444,A -85,B 0,C 180,E1 24683.028,E2 24683.028} C_VEL
LIN {X 0,Y 664.605,Z 408.422,A -85,B 0,C 180,E1 24680.337,E2 24680.337} C_VEL
LIN {X 0,Y 664.597,Z 408.44,A -85,B 0,C 180,E1 24677.151,E2 24677.151} C_VEL
LIN {X 0,Y 664.596,Z 408.418,A -85,B 0,C 180,E1 24674.374,E2 24674.374} C_VEL
LIN {X 0,Y 664.632,Z 408.435,A -85,B 0,C 180,E1 24671.278,E2 24671.278} C_VEL
LIN {X 0,Y 664.596,Z 408.418,A -85,B 0,C 180,E1 24668.392,E2 24668.392} C_VEL
LIN {X 0,Y 664.647,Z 408.435,A -85,B 0,C 180,E1 24665.438,E2 24665.438} C_VEL
LIN {X 0,Y 664.6,Z 408.417,A -85,B 0,C 180,E1 24662.414,E2 24662.414} C_VEL
LIN {X 0,Y 664.646,Z 408.438,A -85,B 0,C 180,E1 24659.483,E2 24659.483} C_VEL
LIN {X 0,Y 664.612,Z 408.415,A -85,B 0,C 180,E1 24656.464,E2 24656.464} C_VEL
LIN {X 0,Y 664.645,Z 408.439,A -85,B 0,C 180,E1 24653.435,E2 24653.435} C_VEL
LIN {X 0,Y 664.623,Z 408.415,A -85,B 0,C 180,E1 24650.387,E2 24650.387} C_VEL
LIN {X 0,Y 664.641,Z 408.437,A -85,B 0,C 180,E1 24647.312,E2 24647.312} C_VEL
LIN {X 0,Y 664.629,Z 408.421,A -85,B 0,C 180,E1 24644.199,E2 24644.199} C_VEL
LIN {X 0,Y 664.635,Z 408.431,A -85,B 0,C 180,E1 24641.128,E2 24641.128} C_VEL
LIN {X 0,Y 664.638,Z 408.43,A -85,B 0,C 180,E1 24638.093,E2 24638.093} C_VEL
LIN {X 0,Y 664.629,Z 408.419,A -85,B 0,C 180,E1 24634.992,E2 24634.992} C_VEL
LIN {X 0,Y 664.644,Z 408.437,A -85,B 0,C 180,E1 24631.909,E2 24631.909} C_VEL
LIN {X 0,Y 664.624,Z 408.43,A -85,B 0,C 180,E1 24628.833,E2 24628.833} C_VEL
LIN {X 0,Y 664.647,Z 408.417,A -85,B 0,C 180,E1 24625.761,E2 24625.761} C_VEL
LIN {X 0,Y 664.642,Z 408.442,A -85,B 0,C 180,E1 24623.517,E2 24623.517} C_VEL
LIN {X 0,Y 663.648,Z 408.567,A -85,B 0,C 180,E1 24622.853,E2 24622.853} C_VEL
LIN {X 0,Y 657.211,Z 409.352,A -85,B 0,C 180,E1 24620.991,E2 24620.991} C_VEL
LIN {X 0,Y 656.671,Z 409.429,A -85,B 0,C 180,E1 24620.507,E2 24620.507} C_VEL
LIN {X 0,Y 656.695,Z 409.55,A -85,B 0,C 180,E1 24620,E2 24620} C_VEL
LIN {X 0,Y 658.07,Z 412.982,A -85,B 0,C 180,E1 24619.549,E2 24619.549} C_VEL
LIN {X 0,Y 659.044,Z 414.907,A -85,B 0,C 180,E1 24619.278,E2 24619.278} C_VEL
LIN {X 0,Y 660.992,Z 418.662,A -85,B 0,C 180,E1 24618.792,E2 24618.792} C_VEL
LIN {X 0,Y 664.361,Z 423.272,A -85,B 0,C 180,E1 24618.386,E2 24618.386} C_VEL
LIN {X 0,Y 680.841,Z 447.322,A -85,B 0,C 180,E1 24616.481,E2 24616.481} C_VEL
LIN {X 0,Y 683.762,Z 452.076,A -85,B 0,C 180,E1 24616.153,E2 24616.153} C_VEL
LIN {X 0,Y 680.664,Z 658.557,A -85,B 0,C 180,E1 24613.409,E2 24613.409} C_VEL
LIN {X 0,Y 677.526,Z 884.674,A -85,B 0,C 180,E1 24610.492,E2 24610.492} C_VEL
LIN {X 0,Y 676.781,Z 910.642,A -85,B 0,C 180,E1 24610.081,E2 24610.081} C_VEL
LIN {X 0,Y 675.855,Z 934.459,A -85,B 0,C 180,E1 24609.575,E2 24609.575} C_VEL
LIN {X 0,Y 674.64,Z 960.881,A -85,B 0,C 180,E1 24608.855,E2 24608.855} C_VEL
LIN {X 0,Y 673.217,Z 985.91,A -85,B 0,C 180,E1 24607.999,E2 24607.999} C_VEL
LIN {X 0,Y 671.918,Z 1006.618,A -85,B 0,C 180,E1 24607.17,E2 24607.17} C_VEL
LIN {X 0,Y 670.496,Z 1027.835,A -85,B 0,C 180,E1 24606.197,E2 24606.197} C_VEL
LIN {X 0,Y 668.882,Z 1050.72,A -85,B 0,C 180,E1 24604.996,E2 24604.996} C_VEL
LIN {X 0,Y 666.965,Z 1075.661,A -85,B 0,C 180,E1 24603.484,E2 24603.484} C_VEL
LIN {X 0,Y 665.442,Z 1095.293,A -85,B 0,C 180,E1 24602.136,E2 24602.136} C_VEL
LIN {X 0,Y 663.9,Z 1115.992,A -85,B 0,C 180,E1 24600.547,E2 24600.547} C_VEL
LIN {X 0,Y 662.293,Z 1137.287,A -85,B 0,C 180,E1 24598.693,E2 24598.693} C_VEL
LIN {X 0,Y 661.067,Z 1153.867,A -85,B 0,C 180,E1 24597.084,E2 24597.084} C_VEL
LIN {X 0,Y 659.907,Z 1171.353,A -85,B 0,C 180,E1 24595.201,E2 24595.201} C_VEL
LIN {X 0,Y 658.761,Z 1188.918,A -85,B 0,C 180,E1 24593.056,E2 24593.056} C_VEL
LIN {X 0,Y 658.014,Z 1202.431,A -85,B 0,C 180,E1 24591.203,E2 24591.203} C_VEL
LIN {X 0,Y 657.323,Z 1216.74,A -85,B 0,C 180,E1 24588.999,E2 24588.999} C_VEL
LIN {X 0,Y 656.749,Z 1229.439,A -85,B 0,C 180,E1 24586.725,E2 24586.725} C_VEL
LIN {X 0,Y 656.463,Z 1238.682,A -85,B 0,C 180,E1 24584.828,E2 24584.828} C_VEL
LIN {X 0,Y 656.232,Z 1247.038,A -85,B 0,C 180,E1 24582.855,E2 24582.855} C_VEL
LIN {X 0,Y 656.058,Z 1255.61,A -85,B 0,C 180,E1 24580.451,E2 24580.451} C_VEL
LIN {X 0,Y 655.943,Z 1262.222,A -85,B 0,C 180,E1 24578.064,E2 24578.064} C_VEL
LIN {X 0,Y 655.928,Z 1266.802,A -85,B 0,C 180,E1 24575.864,E2 24575.864} C_VEL
LIN {X 0,Y 655.914,Z 1270.141,A -85,B 0,C 180,E1 24573.498,E2 24573.498} C_VEL
LIN {X 0,Y 655.89,Z 1271.702,A -85,B 0,C 180,E1 24571.138,E2 24571.138} C_VEL
LIN {X 0,Y 655.863,Z 1271.839,A -85,B 0,C 180,E1 24569.304,E2 24569.304} C_VEL
LIN {X 0,Y 655.904,Z 1270.984,A -85,B 0,C 180,E1 24567.469,E2 24567.469} C_VEL
LIN {X 0,Y 655.911,Z 1268.973,A -85,B 0,C 180,E1 24565.456,E2 24565.456} C_VEL
LIN {X 0,Y 655.932,Z 1265.172,A -85,B 0,C 180,E1 24563.174,E2 24563.174} C_VEL
LIN {X 0,Y 655.95,Z 1259.722,A -85,B 0,C 180,E1 24560.881,E2 24560.881} C_VEL
LIN {X 0,Y 656.068,Z 1253.522,A -85,B 0,C 180,E1 24558.843,E2 24558.843} C_VEL
LIN {X 0,Y 656.24,Z 1246.347,A -85,B 0,C 180,E1 24556.881,E2 24556.881} C_VEL
LIN {X 0,Y 656.472,Z 1238.049,A -85,B 0,C 180,E1 24554.943,E2 24554.943} C_VEL
LIN {X 0,Y 656.879,Z 1227.13,A -85,B 0,C 180,E1 24552.736,E2 24552.736} C_VEL
LIN {X 0,Y 657.449,Z 1213.89,A -85,B 0,C 180,E1 24550.456,E2 24550.456} C_VEL
LIN {X 0,Y 658.082,Z 1201.154,A -85,B 0,C 180,E1 24548.524,E2 24548.524} C_VEL
LIN {X 0,Y 658.955,Z 1186.082,A -85,B 0,C 180,E1 24546.484,E2 24546.484} C_VEL
LIN {X 0,Y 660.034,Z 1168.813,A -85,B 0,C 180,E1 24544.426,E2 24544.426} C_VEL
LIN {X 0,Y 661.16,Z 1152.652,A -85,B 0,C 180,E1 24542.703,E2 24542.703} C_VEL
LIN {X 0,Y 662.576,Z 1133.886,A -85,B 0,C 180,E1 24540.9,E2 24540.9} C_VEL
LIN {X 0,Y 664.134,Z 1112.432,A -85,B 0,C 180,E1 24539.079,E2 24539.079} C_VEL
LIN {X 0,Y 665.557,Z 1093.885,A -85,B 0,C 180,E1 24537.672,E2 24537.672} C_VEL
LIN {X 0,Y 667.237,Z 1072.626,A -85,B 0,C 180,E1 24536.228,E2 24536.228} C_VEL
LIN {X 0,Y 669.049,Z 1048.172,A -85,B 0,C 180,E1 24534.774,E2 24534.774} C_VEL
LIN {X 0,Y 670.569,Z 1026.638,A -85,B 0,C 180,E1 24533.655,E2 24533.655} C_VEL
LIN {X 0,Y 671.995,Z 1005.255,A -85,B 0,C 180,E1 24532.68,E2 24532.68} C_VEL
LIN {X 0,Y 673.627,Z 979.075,A -85,B 0,C 180,E1 24531.656,E2 24531.656} C_VEL
LIN {X 0,Y 675.003,Z 953.04,A -85,B 0,C 180,E1 24530.827,E2 24530.827} C_VEL
LIN {X 0,Y 676.063,Z 929.593,A -85,B 0,C 180,E1 24530.222,E2 24530.222} C_VEL
LIN {X 0,Y 677.075,Z 902.491,A -85,B 0,C 180,E1 24529.68,E2 24529.68} C_VEL
LIN {X 0,Y 677.85,Z 861.664,A -85,B 0,C 180,E1 24529.124,E2 24529.124} C_VEL
LIN {X 0,Y 680.95,Z 639.252,A -85,B 0,C 180,E1 24526.249,E2 24526.249} C_VEL
LIN {X 0,Y 683.766,Z 451.841,A -85,B 0,C 180,E1 24523.754,E2 24523.754} C_VEL
LIN {X 0,Y 670.271,Z 431.81,A -85,B 0,C 180,E1 24522.225,E2 24522.225} C_VEL
LIN {X 0,Y 663.177,Z 421.981,A -85,B 0,C 180,E1 24521.387,E2 24521.387} C_VEL
LIN {X 0,Y 660.621,Z 417.987,A -85,B 0,C 180,E1 24521.063,E2 24521.063} C_VEL
LIN {X 0,Y 658.755,Z 413.91,A -85,B 0,C 180,E1 24520.515,E2 24520.515} C_VEL
LIN {X 0,Y 656.96,Z 410.79,A -85,B 0,C 180,E1 24520.05,E2 24520.05} C_VEL
LIN {X 0,Y 656.655,Z 409.438,A -85,B 0,C 180,E1 24519.871,E2 24519.871} C_VEL
LIN {X 0,Y 656.648,Z 409.432,A -85,B 0,C 180,E1 24517.194,E2 24517.194} C_VEL
LIN {X 0,Y 656.695,Z 409.406,A -85,B 0,C 180,E1 24514.078,E2 24514.078} C_VEL
LIN {X 0,Y 656.64,Z 409.429,A -85,B 0,C 180,E1 24511.282,E2 24511.282} C_VEL
LIN {X 0,Y 656.685,Z 409.424,A -85,B 0,C 180,E1 24508.463,E2 24508.463} C_VEL
LIN {X 0,Y 656.644,Z 409.406,A -85,B 0,C 180,E1 24505.334,E2 24505.334} C_VEL
LIN {X 0,Y 656.643,Z 409.435,A -85,B 0,C 180,E1 24502.659,E2 24502.659} C_VEL
LIN {X 0,Y 656.691,Z 409.411,A -85,B 0,C 180,E1 24499.571,E2 24499.571} C_VEL
LIN {X 0,Y 656.632,Z 409.432,A -85,B 0,C 180,E1 24496.726,E2 24496.726} C_VEL
LIN {X 0,Y 656.68,Z 409.406,A -85,B 0,C 180,E1 24493.921,E2 24493.921} C_VEL
LIN {X 0,Y 656.643,Z 409.427,A -85,B 0,C 180,E1 24490.867,E2 24490.867} C_VEL
LIN {X 0,Y 656.632,Z 409.408,A -85,B 0,C 180,E1 24488.23,E2 24488.23} C_VEL
LIN {X 0,Y 656.706,Z 409.425,A -85,B 0,C 180,E1 24485.242,E2 24485.242} C_VEL
LIN {X 0,Y 656.627,Z 409.41,A -85,B 0,C 180,E1 24482.356,E2 24482.356} C_VEL
LIN {X 0,Y 656.641,Z 409.434,A -85,B 0,C 180,E1 24479.738,E2 24479.738} C_VEL
LIN {X 0,Y 656.658,Z 409.405,A -85,B 0,C 180,E1 24476.595,E2 24476.595} C_VEL
LIN {X 0,Y 656.624,Z 409.434,A -85,B 0,C 180,E1 24473.868,E2 24473.868} C_VEL
LIN {X 0,Y 656.665,Z 409.409,A -85,B 0,C 180,E1 24471.153,E2 24471.153} C_VEL
LIN {X 0,Y 656.634,Z 409.433,A -85,B 0,C 180,E1 24468.048,E2 24468.048} C_VEL
LIN {X 0,Y 656.617,Z 409.418,A -85,B 0,C 180,E1 24465.538,E2 24465.538} C_VEL
LIN {X 0,Y 656.682,Z 409.426,A -85,B 0,C 180,E1 24462.728,E2 24462.728} C_VEL
LIN {X 0,Y 656.621,Z 409.405,A -85,B 0,C 180,E1 24459.684,E2 24459.684} C_VEL
LIN {X 0,Y 656.618,Z 409.434,A -85,B 0,C 180,E1 24457.15,E2 24457.15} C_VEL
LIN {X 0,Y 656.697,Z 409.406,A -85,B 0,C 180,E1 24454.185,E2 24454.185} C_VEL
LIN {X 0,Y 656.615,Z 409.432,A -85,B 0,C 180,E1 24451.288,E2 24451.288} C_VEL
LIN {X 0,Y 656.616,Z 409.429,A -85,B 0,C 180,E1 24448.818,E2 24448.818} C_VEL
LIN {X 0,Y 656.692,Z 409.408,A -85,B 0,C 180,E1 24445.816,E2 24445.816} C_VEL
LIN {X 0,Y 656.611,Z 409.436,A -85,B 0,C 180,E1 24442.913,E2 24442.913} C_VEL
LIN {X 0,Y 656.624,Z 409.55,A -85,B 0,C 180,E1 24440.835,E2 24440.835} C_VEL
LIN {X 0,Y 658.001,Z 413.036,A -85,B 0,C 180,E1 24440.385,E2 24440.385} C_VEL
LIN {X 0,Y 659.127,Z 415.194,A -85,B 0,C 180,E1 24440.082,E2 24440.082} C_VEL
LIN {X 0,Y 665.399,Z 428.061,A -85,B 0,C 180,E1 24438.408,E2 24438.408} C_VEL
LIN {X 0,Y 680.554,Z 450.056,A -85,B 0,C 180,E1 24436.661,E2 24436.661} C_VEL
LIN {X 0,Y 683.476,Z 454.918,A -85,B 0,C 180,E1 24436.329,E2 24436.329} C_VEL
LIN {X 0,Y 683.802,Z 457.514,A -85,B 0,C 180,E1 24436.262,E2 24436.262} C_VEL
LIN {X 0,Y 680.833,Z 657.041,A -85,B 0,C 180,E1 24433.604,E2 24433.604} C_VEL
LIN {X 0,Y 677.716,Z 881.871,A -85,B 0,C 180,E1 24430.701,E2 24430.701} C_VEL
LIN {X 0,Y 676.951,Z 916.055,A -85,B 0,C 180,E1 24430.212,E2 24430.212} C_VEL
LIN {X 0,Y 675.995,Z 941.149,A -85,B 0,C 180,E1 24429.697,E2 24429.697} C_VEL
LIN {X 0,Y 674.914,Z 964.974,A -85,B 0,C 180,E1 24429.073,E2 24429.073} C_VEL
LIN {X 0,Y 673.369,Z 993.275,A -85,B 0,C 180,E1 24428.145,E2 24428.145} C_VEL
LIN {X 0,Y 671.949,Z 1016.053,A -85,B 0,C 180,E1 24427.24,E2 24427.24} C_VEL
LIN {X 0,Y 670.559,Z 1036.791,A -85,B 0,C 180,E1 24426.292,E2 24426.292} C_VEL
LIN {X 0,Y 669.029,Z 1058.499,A -85,B 0,C 180,E1 24425.163,E2 24425.163} C_VEL
LIN {X 0,Y 667.165,Z 1083.455,A -85,B 0,C 180,E1 24423.673,E2 24423.673} C_VEL
LIN {X 0,Y 665.545,Z 1104.029,A -85,B 0,C 180,E1 24422.272,E2 24422.272} C_VEL
LIN {X 0,Y 664.102,Z 1122.917,A -85,B 0,C 180,E1 24420.837,E2 24420.837} C_VEL
LIN {X 0,Y 662.501,Z 1144.761,A -85,B 0,C 180,E1 24418.974,E2 24418.974} C_VEL
LIN {X 0,Y 661.131,Z 1163.014,A -85,B 0,C 180,E1 24417.216,E2 24417.216} C_VEL
LIN {X 0,Y 660.012,Z 1179.263,A -85,B 0,C 180,E1 24415.479,E2 24415.479} C_VEL
LIN {X 0,Y 658.879,Z 1197.166,A -85,B 0,C 180,E1 24413.33,E2 24413.33} C_VEL
LIN {X 0,Y 658.064,Z 1211.488,A -85,B 0,C 180,E1 24411.383,E2 24411.383} C_VEL
LIN {X 0,Y 657.437,Z 1224.223,A -85,B 0,C 180,E1 24409.446,E2 24409.446} C_VEL
LIN {X 0,Y 656.812,Z 1238.297,A -85,B 0,C 180,E1 24406.992,E2 24406.992} C_VEL
LIN {X 0,Y 656.466,Z 1248.499,A -85,B 0,C 180,E1 24404.913,E2 24404.913} C_VEL
LIN {X 0,Y 656.235,Z 1256.882,A -85,B 0,C 180,E1 24402.94,E2 24402.94} C_VEL
LIN {X 0,Y 656.053,Z 1264.884,A -85,B 0,C 180,E1 24400.713,E2 24400.713} C_VEL
LIN {X 0,Y 655.953,Z 1272.132,A -85,B 0,C 180,E1 24398.147,E2 24398.147} C_VEL
LIN {X 0,Y 655.929,Z 1276.734,A -85,B 0,C 180,E1 24395.947,E2 24395.947} C_VEL
LIN {X 0,Y 655.913,Z 1280.097,A -85,B 0,C 180,E1 24393.581,E2 24393.581} C_VEL
LIN {X 0,Y 655.891,Z 1281.693,A -85,B 0,C 180,E1 24391.22,E2 24391.22} C_VEL
LIN {X 0,Y 655.864,Z 1281.849,A -85,B 0,C 180,E1 24389.386,E2 24389.386} C_VEL
LIN {X 0,Y 655.907,Z 1281.012,A -85,B 0,C 180,E1 24387.551,E2 24387.551} C_VEL
LIN {X 0,Y 655.914,Z 1279.021,A -85,B 0,C 180,E1 24385.539,E2 24385.539} C_VEL
LIN {X 0,Y 655.933,Z 1275.246,A -85,B 0,C 180,E1 24383.257,E2 24383.257} C_VEL
LIN {X 0,Y 655.953,Z 1269.832,A -85,B 0,C 180,E1 24380.965,E2 24380.965} C_VEL
LIN {X 0,Y 656.074,Z 1263.351,A -85,B 0,C 180,E1 24378.838,E2 24378.838} C_VEL
LIN {X 0,Y 656.239,Z 1256.503,A -85,B 0,C 180,E1 24376.966,E2 24376.966} C_VEL
LIN {X 0,Y 656.474,Z 1248.065,A -85,B 0,C 180,E1 24374.992,E2 24374.992} C_VEL
LIN {X 0,Y 656.889,Z 1236.876,A -85,B 0,C 180,E1 24372.731,E2 24372.731} C_VEL
LIN {X 0,Y 657.464,Z 1223.58,A -85,B 0,C 180,E1 24370.451,E2 24370.451} C_VEL
LIN {X 0,Y 658.102,Z 1210.807,A -85,B 0,C 180,E1 24368.519,E2 24368.519} C_VEL
LIN {X 0,Y 659.037,Z 1194.992,A -85,B 0,C 180,E1 24366.387,E2 24366.387} C_VEL
LIN {X 0,Y 660.114,Z 1177.505,A -85,B 0,C 180,E1 24364.325,E2 24364.325} C_VEL
LIN {X 0,Y 661.252,Z 1161.506,A -85,B 0,C 180,E1 24362.632,E2 24362.632} C_VEL
LIN {X 0,Y 662.768,Z 1141.081,A -85,B 0,C 180,E1 24360.693,E2 24360.693} C_VEL
LIN {X 0,Y 664.19,Z 1121.697,A -85,B 0,C 180,E1 24359.066,E2 24359.066} C_VEL
LIN {X 0,Y 665.613,Z 1103.214,A -85,B 0,C 180,E1 24357.669,E2 24357.669} C_VEL
LIN {X 0,Y 667.428,Z 1080.424,A -85,B 0,C 180,E1 24356.129,E2 24356.129} C_VEL
LIN {X 0,Y 669.163,Z 1056.412,A -85,B 0,C 180,E1 24354.722,E2 24354.722} C_VEL
LIN {X 0,Y 670.63,Z 1035.673,A -85,B 0,C 180,E1 24353.653,E2 24353.653} C_VEL
LIN {X 0,Y 672.138,Z 1013.047,A -85,B 0,C 180,E1 24352.63,E2 24352.63} C_VEL
LIN {X 0,Y 673.794,Z 985.654,A -85,B 0,C 180,E1 24351.586,E2 24351.586} C_VEL
LIN {X 0,Y 675.051,Z 961.958,A -85,B 0,C 180,E1 24350.841,E2 24350.841} C_VEL
LIN {X 0,Y 676.122,Z 938.177,A -85,B 0,C 180,E1 24350.233,E2 24350.233} C_VEL
LIN {X 0,Y 677.136,Z 910.336,A -85,B 0,C 180,E1 24349.69,E2 24349.69} C_VEL
LIN {X 0,Y 677.974,Z 862.188,A -85,B 0,C 180,E1 24349.048,E2 24349.048} C_VEL
LIN {X 0,Y 681.083,Z 640.165,A -85,B 0,C 180,E1 24346.175,E2 24346.175} C_VEL
LIN {X 0,Y 683.818,Z 456.226,A -85,B 0,C 180,E1 24343.72,E2 24343.72} C_VEL
LIN {X 0,Y 682.825,Z 453.513,A -85,B 0,C 180,E1 24343.593,E2 24343.593} C_VEL
LIN {X 0,Y 672.652,Z 438.564,A -85,B 0,C 180,E1 24342.444,E2 24342.444} C_VEL
LIN {X 0,Y 664.93,Z 427.169,A -85,B 0,C 180,E1 24341.507,E2 24341.507} C_VEL
LIN {X 0,Y 659.745,Z 416.572,A -85,B 0,C 180,E1 24340.1,E2 24340.1} C_VEL
LIN {X 0,Y 658.153,Z 413.249,A -85,B 0,C 180,E1 24339.649,E2 24339.649} C_VEL
LIN {X 0,Y 656.662,Z 409.788,A -85,B 0,C 180,E1 24339.19,E2 24339.19} C_VEL
LIN {X 0,Y 656.614,Z 409.435,A -85,B 0,C 180,E1 24339.083,E2 24339.083} C_VEL
LIN {X 0,Y 656.678,Z 409.436,A -85,B 0,C 180,E1 24336.047,E2 24336.047} C_VEL
LIN {X 0,Y 656.618,Z 409.425,A -85,B 0,C 180,E1 24333.244,E2 24333.244} C_VEL
LIN {X 0,Y 656.656,Z 409.416,A -85,B 0,C 180,E1 24330.57,E2 24330.57} C_VEL
LIN {X 0,Y 656.641,Z 409.433,A -85,B 0,C 180,E1 24327.408,E2 24327.408} C_VEL
LIN {X 0,Y 656.635,Z 409.411,A -85,B 0,C 180,E1 24324.756,E2 24324.756} C_VEL
LIN {X 0,Y 656.703,Z 409.417,A -85,B 0,C 180,E1 24321.715,E2 24321.715} C_VEL
LIN {X 0,Y 656.64,Z 409.425,A -85,B 0,C 180,E1 24318.834,E2 24318.834} C_VEL
LIN {X 0,Y 656.706,Z 409.408,A -85,B 0,C 180,E1 24315.906,E2 24315.906} C_VEL
LIN {X 0,Y 656.654,Z 409.427,A -85,B 0,C 180,E1 24312.845,E2 24312.845} C_VEL
LIN {X 0,Y 656.696,Z 409.406,A -85,B 0,C 180,E1 24309.907,E2 24309.907} C_VEL
LIN {X 0,Y 656.668,Z 409.427,A -85,B 0,C 180,E1 24306.821,E2 24306.821} C_VEL
LIN {X 0,Y 656.694,Z 409.406,A -85,B 0,C 180,E1 24303.841,E2 24303.841} C_VEL
LIN {X 0,Y 656.678,Z 409.426,A -85,B 0,C 180,E1 24300.698,E2 24300.698} C_VEL
LIN {X 0,Y 656.701,Z 409.403,A -85,B 0,C 180,E1 24297.644,E2 24297.644} C_VEL
LIN {X 0,Y 656.682,Z 409.425,A -85,B 0,C 180,E1 24294.495,E2 24294.495} C_VEL
LIN {X 0,Y 656.704,Z 409.403,A -85,B 0,C 180,E1 24291.507,E2 24291.507} C_VEL
LIN {X 0,Y 656.69,Z 409.425,A -85,B 0,C 180,E1 24288.316,E2 24288.316} C_VEL
LIN {X 0,Y 656.699,Z 409.403,A -85,B 0,C 180,E1 24285.269,E2 24285.269} C_VEL
LIN {X 0,Y 656.696,Z 409.426,A -85,B 0,C 180,E1 24282.179,E2 24282.179} C_VEL
LIN {X 0,Y 656.696,Z 409.407,A -85,B 0,C 180,E1 24279.127,E2 24279.127} C_VEL
LIN {X 0,Y 656.701,Z 409.424,A -85,B 0,C 180,E1 24276.002,E2 24276.002} C_VEL
LIN {X 0,Y 656.689,Z 409.426,A -85,B 0,C 180,E1 24272.918,E2 24272.918} C_VEL
LIN {X 0,Y 656.702,Z 409.403,A -85,B 0,C 180,E1 24269.837,E2 24269.837} C_VEL
LIN {X 0,Y 656.681,Z 409.419,A -85,B 0,C 180,E1 24266.76,E2 24266.76} C_VEL
LIN {X 0,Y 656.706,Z 409.429,A -85,B 0,C 180,E1 24263.68,E2 24263.68} C_VEL
LIN {X 0,Y 656.673,Z 409.426,A -85,B 0,C 180,E1 24260.584,E2 24260.584} C_VEL
LIN {X 0,Y 656.671,Z 409.429,A -85,B 0,C 180,E1 24260.507,E2 24260.507} C_VEL
LIN {X 0,Y 656.737,Z 410.317,A -85,B 0,C 180,E1 24260.145,E2 24260.145} C_VEL
LIN {X 0,Y 657.021,Z 413.157,A -85,B 0,C 180,E1 24259.744,E2 24259.744} C_VEL
LIN {X 0,Y 657.842,Z 418.855,A -85,B 0,C 180,E1 24259.285,E2 24259.285} C_VEL
LIN {X 0,Y 660.413,Z 428.524,A -85,B 0,C 180,E1 24258.708,E2 24258.708} C_VEL
LIN {X 0,Y 663.199,Z 433.491,A -85,B 0,C 180,E1 24258.336,E2 24258.336} C_VEL
LIN {X 0,Y 677.228,Z 454.163,A -85,B 0,C 180,E1 24256.7,E2 24256.7} C_VEL
LIN {X 0,Y 678.15,Z 455.985,A -85,B 0,C 180,E1 24256.59,E2 24256.59} C_VEL
LIN {X 0,Y 674.809,Z 661.33,A -85,B 0,C 180,E1 24253.841,E2 24253.841} C_VEL
LIN {X 0,Y 671.384,Z 886.787,A -85,B 0,C 180,E1 24250.907,E2 24250.907} C_VEL
LIN {X 0,Y 670.615,Z 911.366,A -85,B 0,C 180,E1 24250.511,E2 24250.511} C_VEL
LIN {X 0,Y 669.62,Z 935.128,A -85,B 0,C 180,E1 24249.999,E2 24249.999} C_VEL
LIN {X 0,Y 668.28,Z 961.734,A -85,B 0,C 180,E1 24249.265,E2 24249.265} C_VEL
LIN {X 0,Y 666.789,Z 985.924,A -85,B 0,C 180,E1 24248.432,E2 24248.432} C_VEL
LIN {X 0,Y 665.386,Z 1006.63,A -85,B 0,C 180,E1 24247.598,E2 24247.598} C_VEL
LIN {X 0,Y 663.847,Z 1027.844,A -85,B 0,C 180,E1 24246.618,E2 24246.618} C_VEL
LIN {X 0,Y 662.045,Z 1051.66,A -85,B 0,C 180,E1 24245.356,E2 24245.356} C_VEL
LIN {X 0,Y 660.047,Z 1075.668,A -85,B 0,C 180,E1 24243.882,E2 24243.882} C_VEL
LIN {X 0,Y 658.383,Z 1095.3,A -85,B 0,C 180,E1 24242.523,E2 24242.523} C_VEL
LIN {X 0,Y 656.688,Z 1115.941,A -85,B 0,C 180,E1 24240.924,E2 24240.924} C_VEL
LIN {X 0,Y 654.941,Z 1137.293,A -85,B 0,C 180,E1 24239.046,E2 24239.046} C_VEL
LIN {X 0,Y 653.61,Z 1153.871,A -85,B 0,C 180,E1 24237.419,E2 24237.419} C_VEL
LIN {X 0,Y 652.279,Z 1171.858,A -85,B 0,C 180,E1 24235.459,E2 24235.459} C_VEL
LIN {X 0,Y 651.049,Z 1189.23,A -85,B 0,C 180,E1 24233.304,E2 24233.304} C_VEL
LIN {X 0,Y 650.243,Z 1202.435,A -85,B 0,C 180,E1 24231.469,E2 24231.469} C_VEL
LIN {X 0,Y 649.478,Z 1216.742,A -85,B 0,C 180,E1 24229.238,E2 24229.238} C_VEL
LIN {X 0,Y 648.853,Z 1229.443,A -85,B 0,C 180,E1 24226.935,E2 24226.935} C_VEL
LIN {X 0,Y 648.519,Z 1238.686,A -85,B 0,C 180,E1 24225.014,E2 24225.014} C_VEL
LIN {X 0,Y 648.261,Z 1247.04,A -85,B 0,C 180,E1 24223.016,E2 24223.016} C_VEL
LIN {X 0,Y 648.069,Z 1255.438,A -85,B 0,C 180,E1 24220.637,E2 24220.637} C_VEL
LIN {X 0,Y 647.958,Z 1262.22,A -85,B 0,C 180,E1 24218.164,E2 24218.164} C_VEL
LIN {X 0,Y 647.929,Z 1266.8,A -85,B 0,C 180,E1 24215.937,E2 24215.937} C_VEL
LIN {X 0,Y 647.914,Z 1270.141,A -85,B 0,C 180,E1 24213.541,E2 24213.541} C_VEL
LIN {X 0,Y 647.898,Z 1271.68,A -85,B 0,C 180,E1 24211.241,E2 24211.241} C_VEL
LIN {X 0,Y 647.863,Z 1271.839,A -85,B 0,C 180,E1 24209.295,E2 24209.295} C_VEL
LIN {X 0,Y 647.904,Z 1270.983,A -85,B 0,C 180,E1 24207.438,E2 24207.438} C_VEL
LIN {X 0,Y 647.911,Z 1268.969,A -85,B 0,C 180,E1 24205.4,E2 24205.4} C_VEL
LIN {X 0,Y 647.934,Z 1265.171,A -85,B 0,C 180,E1 24203.089,E2 24203.089} C_VEL
LIN {X 0,Y 647.956,Z 1259.974,A -85,B 0,C 180,E1 24200.857,E2 24200.857} C_VEL
LIN {X 0,Y 648.094,Z 1253.52,A -85,B 0,C 180,E1 24198.704,E2 24198.704} C_VEL
LIN {X 0,Y 648.264,Z 1246.703,A -85,B 0,C 180,E1 24196.808,E2 24196.808} C_VEL
LIN {X 0,Y 648.518,Z 1238.412,A -85,B 0,C 180,E1 24194.835,E2 24194.835} C_VEL
LIN {X 0,Y 648.914,Z 1228.525,A -85,B 0,C 180,E1 24192.795,E2 24192.795} C_VEL
LIN {X 0,Y 649.56,Z 1215.031,A -85,B 0,C 180,E1 24190.396,E2 24190.396} C_VEL
LIN {X 0,Y 650.283,Z 1201.797,A -85,B 0,C 180,E1 24188.348,E2 24188.348} C_VEL
LIN {X 0,Y 651.175,Z 1187.501,A -85,B 0,C 180,E1 24186.378,E2 24186.378} C_VEL
LIN {X 0,Y 652.404,Z 1169.651,A -85,B 0,C 180,E1 24184.202,E2 24184.202} C_VEL
LIN {X 0,Y 653.693,Z 1152.915,A -85,B 0,C 180,E1 24182.393,E2 24182.393} C_VEL
LIN {X 0,Y 655.16,Z 1134.786,A -85,B 0,C 180,E1 24180.628,E2 24180.628} C_VEL
LIN {X 0,Y 656.921,Z 1112.847,A -85,B 0,C 180,E1 24178.737,E2 24178.737} C_VEL
LIN {X 0,Y 658.513,Z 1093.874,A -85,B 0,C 180,E1 24177.284,E2 24177.284} C_VEL
LIN {X 0,Y 660.26,Z 1073.349,A -85,B 0,C 180,E1 24175.874,E2 24175.874} C_VEL
LIN {X 0,Y 662.284,Z 1048.163,A -85,B 0,C 180,E1 24174.36,E2 24174.36} C_VEL
LIN {X 0,Y 663.907,Z 1026.942,A -85,B 0,C 180,E1 24173.248,E2 24173.248} C_VEL
LIN {X 0,Y 665.481,Z 1005.124,A -85,B 0,C 180,E1 24172.246,E2 24172.246} C_VEL
LIN {X 0,Y 667.249,Z 979.06,A -85,B 0,C 180,E1 24171.222,E2 24171.222} C_VEL
LIN {X 0,Y 668.718,Z 953.197,A -85,B 0,C 180,E1 24170.393,E2 24170.393} C_VEL
LIN {X 0,Y 669.846,Z 930.068,A -85,B 0,C 180,E1 24169.791,E2 24169.791} C_VEL
LIN {X 0,Y 670.92,Z 903.494,A -85,B 0,C 180,E1 24169.253,E2 24169.253} C_VEL
LIN {X 0,Y 671.738,Z 865.645,A -85,B 0,C 180,E1 24168.727,E2 24168.727} C_VEL
LIN {X 0,Y 675.103,Z 642.969,A -85,B 0,C 180,E1 24165.827,E2 24165.827} C_VEL
LIN {X 0,Y 678.156,Z 455.622,A -85,B 0,C 180,E1 24163.315,E2 24163.315} C_VEL
LIN {X 0,Y 663.566,Z 433.953,A -85,B 0,C 180,E1 24161.617,E2 24161.617} C_VEL
LIN {X 0,Y 655.255,Z 422.589,A -85,B 0,C 180,E1 24160.604,E2 24160.604} C_VEL
LIN {X 0,Y 652.148,Z 418.13,A -85,B 0,C 180,E1 24160.203,E2 24160.203} C_VEL
LIN {X 0,Y 650.268,Z 414.27,A -85,B 0,C 180,E1 24159.653,E2 24159.653} C_VEL
LIN {X 0,Y 648.792,Z 410.915,A -85,B 0,C 180,E1 24159.184,E2 24159.184} C_VEL
LIN {X 0,Y 648.723,Z 410.42,A -85,B 0,C 180,E1 24159.08,E2 24159.08} C_VEL
LIN {X 0,Y 648.724,Z 410.42,A -85,B 0,C 180,E1 24155.841,E2 24155.841} C_VEL
LIN {X 0,Y 648.706,Z 410.413,A -85,B 0,C 180,E1 24153.069,E2 24153.069} C_VEL
LIN {X 0,Y 648.761,Z 410.391,A -85,B 0,C 180,E1 24149.958,E2 24149.958} C_VEL
LIN {X 0,Y 648.699,Z 410.421,A -85,B 0,C 180,E1 24147.145,E2 24147.145} C_VEL
LIN {X 0,Y 648.745,Z 410.4,A -85,B 0,C 180,E1 24144.3,E2 24144.3} C_VEL
LIN {X 0,Y 648.705,Z 410.407,A -85,B 0,C 180,E1 24141.182,E2 24141.182} C_VEL
LIN {X 0,Y 648.703,Z 410.415,A -85,B 0,C 180,E1 24138.513,E2 24138.513} C_VEL
LIN {X 0,Y 648.756,Z 410.389,A -85,B 0,C 180,E1 24135.464,E2 24135.464} C_VEL
LIN {X 0,Y 648.693,Z 410.419,A -85,B 0,C 180,E1 24132.643,E2 24132.643} C_VEL
LIN {X 0,Y 648.73,Z 410.399,A -85,B 0,C 180,E1 24129.851,E2 24129.851} C_VEL
LIN {X 0,Y 648.704,Z 410.42,A -85,B 0,C 180,E1 24126.727,E2 24126.727} C_VEL
LIN {X 0,Y 648.693,Z 410.413,A -85,B 0,C 180,E1 24124.066,E2 24124.066} C_VEL
LIN {X 0,Y 648.755,Z 410.412,A -85,B 0,C 180,E1 24120.971,E2 24120.971} C_VEL
LIN {X 0,Y 648.687,Z 410.414,A -85,B 0,C 180,E1 24118.145,E2 24118.145} C_VEL
LIN {X 0,Y 648.716,Z 410.403,A -85,B 0,C 180,E1 24115.403,E2 24115.403} C_VEL
LIN {X 0,Y 648.702,Z 410.412,A -85,B 0,C 180,E1 24112.293,E2 24112.293} C_VEL
LIN {X 0,Y 648.683,Z 410.405,A -85,B 0,C 180,E1 24109.61,E2 24109.61} C_VEL
LIN {X 0,Y 648.769,Z 410.406,A -85,B 0,C 180,E1 24106.633,E2 24106.633} C_VEL
LIN {X 0,Y 648.681,Z 410.412,A -85,B 0,C 180,E1 24103.708,E2 24103.708} C_VEL
LIN {X 0,Y 648.692,Z 410.422,A -85,B 0,C 180,E1 24101.114,E2 24101.114} C_VEL
LIN {X 0,Y 648.722,Z 410.413,A -85,B 0,C 180,E1 24098.004,E2 24098.004} C_VEL
LIN {X 0,Y 648.675,Z 410.411,A -85,B 0,C 180,E1 24095.309,E2 24095.309} C_VEL
LIN {X 0,Y 648.712,Z 410.42,A -85,B 0,C 180,E1 24092.557,E2 24092.557} C_VEL
LIN {X 0,Y 648.686,Z 410.405,A -85,B 0,C 180,E1 24089.425,E2 24089.425} C_VEL
LIN {X 0,Y 648.674,Z 410.418,A -85,B 0,C 180,E1 24086.816,E2 24086.816} C_VEL
LIN {X 0,Y 648.756,Z 410.421,A -85,B 0,C 180,E1 24083.822,E2 24083.822} C_VEL
LIN {X 0,Y 648.748,Z 410.465,A -85,B 0,C 180,E1 24081.601,E2 24081.601} C_VEL
LIN {X 0,Y 649.739,Z 413.5,A -85,B 0,C 180,E1 24081.219,E2 24081.219} C_VEL
LIN {X 0,Y 650.827,Z 415.123,A -85,B 0,C 180,E1 24080.957,E2 24080.957} C_VEL
LIN {X 0,Y 652.702,Z 419.059,A -85,B 0,C 180,E1 24080.41,E2 24080.41} C_VEL
LIN {X 0,Y 657.079,Z 428.005,A -85,B 0,C 180,E1 24079.231,E2 24079.231} C_VEL
LIN {X 0,Y 674.697,Z 453.464,A -85,B 0,C 180,E1 24077.138,E2 24077.138} C_VEL
LIN {X 0,Y 678.238,Z 459.176,A -85,B 0,C 180,E1 24076.73,E2 24076.73} C_VEL
LIN {X 0,Y 675.006,Z 658.956,A -85,B 0,C 180,E1 24074.05,E2 24074.05} C_VEL
LIN {X 0,Y 671.619,Z 883.898,A -85,B 0,C 180,E1 24071.122,E2 24071.122} C_VEL
LIN {X 0,Y 670.785,Z 916.968,A -85,B 0,C 180,E1 24070.638,E2 24070.638} C_VEL
LIN {X 0,Y 669.788,Z 941.389,A -85,B 0,C 180,E1 24070.132,E2 24070.132} C_VEL
LIN {X 0,Y 668.633,Z 964.961,A -85,B 0,C 180,E1 24069.511,E2 24069.511} C_VEL
LIN {X 0,Y 666.957,Z 993.272,A -85,B 0,C 180,E1 24068.578,E2 24068.578} C_VEL
LIN {X 0,Y 665.413,Z 1016.175,A -85,B 0,C 180,E1 24067.663,E2 24067.663} C_VEL
LIN {X 0,Y 663.851,Z 1037.793,A -85,B 0,C 180,E1 24066.665,E2 24066.665} C_VEL
LIN {X 0,Y 662.093,Z 1060.971,A -85,B 0,C 180,E1 24065.439,E2 24065.439} C_VEL
LIN {X 0,Y 660.05,Z 1085.656,A -85,B 0,C 180,E1 24063.929,E2 24063.929} C_VEL
LIN {X 0,Y 658.446,Z 1104.628,A -85,B 0,C 180,E1 24062.617,E2 24062.617} C_VEL
LIN {X 0,Y 656.819,Z 1124.128,A -85,B 0,C 180,E1 24061.115,E2 24061.115} C_VEL
LIN {X 0,Y 654.985,Z 1146.793,A -85,B 0,C 180,E1 24059.138,E2 24059.138} C_VEL
LIN {X 0,Y 653.646,Z 1163.42,A -85,B 0,C 180,E1 24057.51,E2 24057.51} C_VEL
LIN {X 0,Y 652.363,Z 1180.317,A -85,B 0,C 180,E1 24055.678,E2 24055.678} C_VEL
LIN {X 0,Y 651.095,Z 1198.589,A -85,B 0,C 180,E1 24053.433,E2 24053.433} C_VEL
LIN {X 0,Y 650.243,Z 1212.431,A -85,B 0,C 180,E1 24051.515,E2 24051.515} C_VEL
LIN {X 0,Y 649.49,Z 1226.543,A -85,B 0,C 180,E1 24049.314,E2 24049.314} C_VEL
LIN {X 0,Y 648.87,Z 1239.229,A -85,B 0,C 180,E1 24047.021,E2 24047.021} C_VEL
LIN {X 0,Y 648.519,Z 1248.5,A -85,B 0,C 180,E1 24045.1,E2 24045.1} C_VEL
LIN {X 0,Y 648.263,Z 1256.883,A -85,B 0,C 180,E1 24043.102,E2 24043.102} C_VEL
LIN {X 0,Y 648.071,Z 1264.581,A -85,B 0,C 180,E1 24040.936,E2 24040.936} C_VEL
LIN {X 0,Y 647.978,Z 1271.921,A -85,B 0,C 180,E1 24038.337,E2 24038.337} C_VEL
LIN {X 0,Y 647.932,Z 1276.572,A -85,B 0,C 180,E1 24036.11,E2 24036.11} C_VEL
LIN {X 0,Y 647.914,Z 1279.894,A -85,B 0,C 180,E1 24033.802,E2 24033.802} C_VEL
LIN {X 0,Y 647.9,Z 1281.67,A -85,B 0,C 180,E1 24031.324,E2 24031.324} C_VEL
LIN {X 0,Y 647.864,Z 1281.849,A -85,B 0,C 180,E1 24029.378,E2 24029.378} C_VEL
LIN {X 0,Y 647.908,Z 1281.012,A -85,B 0,C 180,E1 24027.521,E2 24027.521} C_VEL
LIN {X 0,Y 647.913,Z 1279.018,A -85,B 0,C 180,E1 24025.484,E2 24025.484} C_VEL
LIN {X 0,Y 647.936,Z 1275.246,A -85,B 0,C 180,E1 24023.173,E2 24023.173} C_VEL
LIN {X 0,Y 647.955,Z 1269.832,A -85,B 0,C 180,E1 24020.852,E2 24020.852} C_VEL
LIN {X 0,Y 648.1,Z 1263.35,A -85,B 0,C 180,E1 24018.699,E2 24018.699} C_VEL
LIN {X 0,Y 648.264,Z 1256.504,A -85,B 0,C 180,E1 24016.802,E2 24016.802} C_VEL
LIN {X 0,Y 648.528,Z 1248.067,A -85,B 0,C 180,E1 24014.803,E2 24014.803} C_VEL
LIN {X 0,Y 648.971,Z 1237.343,A -85,B 0,C 180,E1 24012.607,E2 24012.607} C_VEL
LIN {X 0,Y 649.599,Z 1224.151,A -85,B 0,C 180,E1 24010.298,E2 24010.298} C_VEL
LIN {X 0,Y 650.303,Z 1211.454,A -85,B 0,C 180,E1 24008.343,E2 24008.343} C_VEL
LIN {X 0,Y 651.205,Z 1197.126,A -85,B 0,C 180,E1 24006.373,E2 24006.373} C_VEL
LIN {X 0,Y 652.432,Z 1179.212,A -85,B 0,C 180,E1 24004.198,E2 24004.198} C_VEL
LIN {X 0,Y 653.684,Z 1162.992,A -85,B 0,C 180,E1 24002.446,E2 24002.446} C_VEL
LIN {X 0,Y 655.123,Z 1145.211,A -85,B 0,C 180,E1 24000.713,E2 24000.713} C_VEL
LIN {X 0,Y 656.894,Z 1123.188,A -85,B 0,C 180,E1 23998.81,E2 23998.81} C_VEL
LIN {X 0,Y 658.452,Z 1104.546,A -85,B 0,C 180,E1 23997.378,E2 23997.378} C_VEL
LIN {X 0,Y 660.124,Z 1084.831,A -85,B 0,C 180,E1 23996.017,E2 23996.017} C_VEL
LIN {X 0,Y 662.161,Z 1059.975,A -85,B 0,C 180,E1 23994.505,E2 23994.505} C_VEL
LIN {X 0,Y 663.859,Z 1037.68,A -85,B 0,C 180,E1 23993.329,E2 23993.329} C_VEL
LIN {X 0,Y 665.417,Z 1016.11,A -85,B 0,C 180,E1 23992.334,E2 23992.334} C_VEL
LIN {X 0,Y 667.108,Z 991.198,A -85,B 0,C 180,E1 23991.343,E2 23991.343} C_VEL
LIN {X 0,Y 668.673,Z 964.111,A -85,B 0,C 180,E1 23990.464,E2 23990.464} C_VEL
LIN {X 0,Y 669.811,Z 940.839,A -85,B 0,C 180,E1 23989.855,E2 23989.855} C_VEL
LIN {X 0,Y 670.851,Z 915.34,A -85,B 0,C 180,E1 23989.331,E2 23989.331} C_VEL
LIN {X 0,Y 671.674,Z 880.13,A -85,B 0,C 180,E1 23988.83,E2 23988.83} C_VEL
LIN {X 0,Y 675.049,Z 656.267,A -85,B 0,C 180,E1 23985.915,E2 23985.915} C_VEL
LIN {X 0,Y 678.243,Z 458.854,A -85,B 0,C 180,E1 23983.265,E2 23983.265} C_VEL
LIN {X 0,Y 665.031,Z 439.334,A -85,B 0,C 180,E1 23981.735,E2 23981.735} C_VEL
LIN {X 0,Y 656.475,Z 427.029,A -85,B 0,C 180,E1 23980.666,E2 23980.666} C_VEL
LIN {X 0,Y 652.319,Z 418.538,A -85,B 0,C 180,E1 23979.503,E2 23979.503} C_VEL
LIN {X 0,Y 650.099,Z 414.045,A -85,B 0,C 180,E1 23978.868,E2 23978.868} C_VEL
LIN {X 0,Y 648.889,Z 411.223,A -85,B 0,C 180,E1 23978.483,E2 23978.483} C_VEL
LIN {X 0,Y 648.757,Z 410.396,A -85,B 0,C 180,E1 23978.362,E2 23978.362} C_VEL
LIN {X 0,Y 648.678,Z 410.423,A -85,B 0,C 180,E1 23975.371,E2 23975.371} C_VEL
LIN {X 0,Y 648.699,Z 410.417,A -85,B 0,C 180,E1 23972.754,E2 23972.754} C_VEL
LIN {X 0,Y 648.706,Z 410.401,A -85,B 0,C 180,E1 23969.554,E2 23969.554} C_VEL
LIN {X 0,Y 648.692,Z 410.424,A -85,B 0,C 180,E1 23966.947,E2 23966.947} C_VEL
LIN {X 0,Y 648.773,Z 410.406,A -85,B 0,C 180,E1 23963.912,E2 23963.912} C_VEL
LIN {X 0,Y 648.699,Z 410.404,A -85,B 0,C 180,E1 23960.953,E2 23960.953} C_VEL
LIN {X 0,Y 648.759,Z 410.418,A -85,B 0,C 180,E1 23958.047,E2 23958.047} C_VEL
LIN {X 0,Y 648.712,Z 410.39,A -85,B 0,C 180,E1 23955.008,E2 23955.008} C_VEL
LIN {X 0,Y 648.735,Z 410.42,A -85,B 0,C 180,E1 23952.19,E2 23952.19} C_VEL
LIN {X 0,Y 648.729,Z 410.387,A -85,B 0,C 180,E1 23948.956,E2 23948.956} C_VEL
LIN {X 0,Y 648.743,Z 410.422,A -85,B 0,C 180,E1 23946.016,E2 23946.016} C_VEL
LIN {X 0,Y 648.738,Z 410.387,A -85,B 0,C 180,E1 23942.827,E2 23942.827} C_VEL
LIN {X 0,Y 648.755,Z 410.422,A -85,B 0,C 180,E1 23939.823,E2 23939.823} C_VEL
LIN {X 0,Y 648.745,Z 410.387,A -85,B 0,C 180,E1 23936.642,E2 23936.642} C_VEL
LIN {X 0,Y 648.769,Z 410.418,A -85,B 0,C 180,E1 23933.54,E2 23933.54} C_VEL
LIN {X 0,Y 648.747,Z 410.389,A -85,B 0,C 180,E1 23930.418,E2 23930.418} C_VEL
LIN {X 0,Y 648.763,Z 410.414,A -85,B 0,C 180,E1 23927.315,E2 23927.315} C_VEL
LIN {X 0,Y 648.75,Z 410.397,A -85,B 0,C 180,E1 23924.169,E2 23924.169} C_VEL
LIN {X 0,Y 648.757,Z 410.407,A -85,B 0,C 180,E1 23921.115,E2 23921.115} C_VEL
LIN {X 0,Y 648.757,Z 410.408,A -85,B 0,C 180,E1 23918.005,E2 23918.005} C_VEL
LIN {X 0,Y 648.748,Z 410.392,A -85,B 0,C 180,E1 23914.922,E2 23914.922} C_VEL
LIN {X 0,Y 648.763,Z 410.417,A -85,B 0,C 180,E1 23911.834,E2 23911.834} C_VEL
LIN {X 0,Y 648.746,Z 410.405,A -85,B 0,C 180,E1 23908.804,E2 23908.804} C_VEL
LIN {X 0,Y 648.766,Z 410.392,A -85,B 0,C 180,E1 23905.7,E2 23905.7} C_VEL
LIN {X 0,Y 648.735,Z 410.401,A -85,B 0,C 180,E1 23902.607,E2 23902.607} C_VEL
LIN {X 0,Y 648.749,Z 410.411,A -85,B 0,C 180,E1 23900.777,E2 23900.777} C_VEL
LIN {X 0,Y 649.99,Z 413.838,A -85,B 0,C 180,E1 23900.327,E2 23900.327} C_VEL
LIN {X 0,Y 651.093,Z 415.853,A -85,B 0,C 180,E1 23900.025,E2 23900.025} C_VEL
LIN {X 0,Y 652.671,Z 418.803,A -85,B 0,C 180,E1 23899.635,E2 23899.635} C_VEL
LIN {X 0,Y 663.199,Z 433.491,A -85,B 0,C 180,E1 23898.336,E2 23898.336} C_VEL
LIN {X 0,Y 664.887,Z 436.759,A -85,B 0,C 180,E1 23898.121,E2 23898.121} C_VEL
LIN {X 0,Y 666.477,Z 444.304,A -85,B 0,C 180,E1 23897.849,E2 23897.849} C_VEL
LIN {X 0,Y 667.904,Z 451.276,A -85,B 0,C 180,E1 23897.604,E2 23897.604} C_VEL
LIN {X 0,Y 669.215,Z 454.224,A -85,B 0,C 180,E1 23897.434,E2 23897.434} C_VEL
LIN {X 0,Y 672.582,Z 459.669,A -85,B 0,C 180,E1 23897.038,E2 23897.038} C_VEL
LIN {X 0,Y 668.999,Z 663.693,A -85,B 0,C 180,E1 23894.287,E2 23894.287} C_VEL
LIN {X 0,Y 665.295,Z 888.19,A -85,B 0,C 180,E1 23891.34,E2 23891.34} C_VEL
LIN {X 0,Y 664.499,Z 911.855,A -85,B 0,C 180,E1 23890.952,E2 23890.952} C_VEL
LIN {X 0,Y 663.443,Z 935.374,A -85,B 0,C 180,E1 23890.442,E2 23890.442} C_VEL
LIN {X 0,Y 661.958,Z 962.489,A -85,B 0,C 180,E1 23889.686,E2 23889.686} C_VEL
LIN {X 0,Y 660.364,Z 986.515,A -85,B 0,C 180,E1 23888.85,E2 23888.85} C_VEL
LIN {X 0,Y 658.817,Z 1007.771,A -85,B 0,C 180,E1 23887.984,E2 23887.984} C_VEL
LIN {X 0,Y 657.096,Z 1029.855,A -85,B 0,C 180,E1 23886.947,E2 23886.947} C_VEL
LIN {X 0,Y 654.935,Z 1055.725,A -85,B 0,C 180,E1 23885.537,E2 23885.537} C_VEL
LIN {X 0,Y 653.015,Z 1077.143,A -85,B 0,C 180,E1 23884.192,E2 23884.192} C_VEL
LIN {X 0,Y 651.325,Z 1095.719,A -85,B 0,C 180,E1 23882.887,E2 23882.887} C_VEL
LIN {X 0,Y 649.409,Z 1117.159,A -85,B 0,C 180,E1 23881.207,E2 23881.207} C_VEL
LIN {X 0,Y 647.566,Z 1137.808,A -85,B 0,C 180,E1 23879.358,E2 23879.358} C_VEL
LIN {X 0,Y 646.146,Z 1154.183,A -85,B 0,C 180,E1 23877.729,E2 23877.729} C_VEL
LIN {X 0,Y 644.644,Z 1172.679,A -85,B 0,C 180,E1 23875.687,E2 23875.687} C_VEL
LIN {X 0,Y 643.342,Z 1189.642,A -85,B 0,C 180,E1 23873.544,E2 23873.544} C_VEL
LIN {X 0,Y 642.442,Z 1203.072,A -85,B 0,C 180,E1 23871.647,E2 23871.647} C_VEL
LIN {X 0,Y 641.614,Z 1217.313,A -85,B 0,C 180,E1 23869.388,E2 23869.388} C_VEL
LIN {X 0,Y 640.939,Z 1229.913,A -85,B 0,C 180,E1 23867.057,E2 23867.057} C_VEL
LIN {X 0,Y 640.566,Z 1239.1,A -85,B 0,C 180,E1 23865.112,E2 23865.112} C_VEL
LIN {X 0,Y 640.285,Z 1247.394,A -85,B 0,C 180,E1 23863.089,E2 23863.089} C_VEL
LIN {X 0,Y 640.078,Z 1255.872,A -85,B 0,C 180,E1 23860.624,E2 23860.624} C_VEL
LIN {X 0,Y 639.961,Z 1262.425,A -85,B 0,C 180,E1 23858.176,E2 23858.176} C_VEL
LIN {X 0,Y 639.93,Z 1266.958,A -85,B 0,C 180,E1 23855.921,E2 23855.921} C_VEL
LIN {X 0,Y 639.913,Z 1270.232,A -85,B 0,C 180,E1 23853.496,E2 23853.496} C_VEL
LIN {X 0,Y 639.891,Z 1271.702,A -85,B 0,C 180,E1 23851.166,E2 23851.166} C_VEL
LIN {X 0,Y 639.863,Z 1271.839,A -85,B 0,C 180,E1 23849.286,E2 23849.286} C_VEL
LIN {X 0,Y 639.905,Z 1270.983,A -85,B 0,C 180,E1 23847.406,E2 23847.406} C_VEL
LIN {X 0,Y 639.912,Z 1268.965,A -85,B 0,C 180,E1 23845.342,E2 23845.342} C_VEL
LIN {X 0,Y 639.939,Z 1265.17,A -85,B 0,C 180,E1 23843.003,E2 23843.003} C_VEL
LIN {X 0,Y 639.962,Z 1259.972,A -85,B 0,C 180,E1 23840.742,E2 23840.742} C_VEL
LIN {X 0,Y 640.121,Z 1253.517,A -85,B 0,C 180,E1 23838.561,E2 23838.561} C_VEL
LIN {X 0,Y 640.291,Z 1246.658,A -85,B 0,C 180,E1 23836.629,E2 23836.629} C_VEL
LIN {X 0,Y 640.568,Z 1238.701,A -85,B 0,C 180,E1 23834.708,E2 23834.708} C_VEL
LIN {X 0,Y 641,Z 1228.989,A -85,B 0,C 180,E1 23832.67,E2 23832.67} C_VEL
LIN {X 0,Y 641.696,Z 1215.598,A -85,B 0,C 180,E1 23830.241,E2 23830.241} C_VEL
LIN {X 0,Y 642.487,Z 1202.432,A -85,B 0,C 180,E1 23828.168,E2 23828.168} C_VEL
LIN {X 0,Y 643.406,Z 1188.812,A -85,B 0,C 180,E1 23826.255,E2 23826.255} C_VEL
LIN {X 0,Y 644.727,Z 1171.334,A -85,B 0,C 180,E1 23824.07,E2 23824.07} C_VEL
LIN {X 0,Y 646.179,Z 1153.834,A -85,B 0,C 180,E1 23822.144,E2 23822.144} C_VEL
LIN {X 0,Y 647.619,Z 1137.242,A -85,B 0,C 180,E1 23820.498,E2 23820.498} C_VEL
LIN {X 0,Y 649.508,Z 1115.865,A -85,B 0,C 180,E1 23818.598,E2 23818.598} C_VEL
LIN {X 0,Y 651.311,Z 1095.866,A -85,B 0,C 180,E1 23817.033,E2 23817.033} C_VEL
LIN {X 0,Y 653.027,Z 1077.011,A -85,B 0,C 180,E1 23815.709,E2 23815.709} C_VEL
LIN {X 0,Y 655.001,Z 1055.074,A -85,B 0,C 180,E1 23814.333,E2 23814.333} C_VEL
LIN {X 0,Y 657.112,Z 1029.617,A -85,B 0,C 180,E1 23812.951,E2 23812.951} C_VEL
LIN {X 0,Y 658.754,Z 1008.611,A -85,B 0,C 180,E1 23811.963,E2 23811.963} C_VEL
LIN {X 0,Y 660.337,Z 986.874,A -85,B 0,C 180,E1 23811.073,E2 23811.073} C_VEL
LIN {X 0,Y 662.037,Z 961.325,A -85,B 0,C 180,E1 23810.186,E2 23810.186} C_VEL
LIN {X 0,Y 663.486,Z 934.403,A -85,B 0,C 180,E1 23809.445,E2 23809.445} C_VEL
LIN {X 0,Y 664.527,Z 911.027,A -85,B 0,C 180,E1 23808.942,E2 23808.942} C_VEL
LIN {X 0,Y 665.359,Z 886.032,A -85,B 0,C 180,E1 23808.539,E2 23808.539} C_VEL
LIN {X 0,Y 669.032,Z 661.758,A -85,B 0,C 180,E1 23805.597,E2 23805.597} C_VEL
LIN {X 0,Y 672.585,Z 459.372,A -85,B 0,C 180,E1 23802.868,E2 23802.868} C_VEL
LIN {X 0,Y 658.802,Z 439.024,A -85,B 0,C 180,E1 23801.23,E2 23801.23} C_VEL
LIN {X 0,Y 648.017,Z 424.053,A -85,B 0,C 180,E1 23799.875,E2 23799.875} C_VEL
LIN {X 0,Y 643.612,Z 418.076,A -85,B 0,C 180,E1 23799.278,E2 23799.278} C_VEL
LIN {X 0,Y 642.291,Z 415.142,A -85,B 0,C 180,E1 23798.857,E2 23798.857} C_VEL
LIN {X 0,Y 640.84,Z 411.479,A -85,B 0,C 180,E1 23798.346,E2 23798.346} C_VEL
LIN {X 0,Y 640.763,Z 411.399,A -85,B 0,C 180,E1 23795.376,E2 23795.376} C_VEL
LIN {X 0,Y 640.831,Z 411.406,A -85,B 0,C 180,E1 23792.431,E2 23792.431} C_VEL
LIN {X 0,Y 640.768,Z 411.389,A -85,B 0,C 180,E1 23789.442,E2 23789.442} C_VEL
LIN {X 0,Y 640.768,Z 411.404,A -85,B 0,C 180,E1 23786.806,E2 23786.806} C_VEL
LIN {X 0,Y 640.807,Z 411.407,A -85,B 0,C 180,E1 23783.642,E2 23783.642} C_VEL
LIN {X 0,Y 640.755,Z 411.389,A -85,B 0,C 180,E1 23780.83,E2 23780.83} C_VEL
LIN {X 0,Y 640.83,Z 411.407,A -85,B 0,C 180,E1 23777.881,E2 23777.881} C_VEL
LIN {X 0,Y 640.753,Z 411.378,A -85,B 0,C 180,E1 23774.828,E2 23774.828} C_VEL
LIN {X 0,Y 640.771,Z 411.41,A -85,B 0,C 180,E1 23772.161,E2 23772.161} C_VEL
LIN {X 0,Y 640.77,Z 411.377,A -85,B 0,C 180,E1 23768.887,E2 23768.887} C_VEL
LIN {X 0,Y 640.752,Z 411.411,A -85,B 0,C 180,E1 23766.271,E2 23766.271} C_VEL
LIN {X 0,Y 640.823,Z 411.375,A -85,B 0,C 180,E1 23763.31,E2 23763.31} C_VEL
LIN {X 0,Y 640.756,Z 411.41,A -85,B 0,C 180,E1 23760.358,E2 23760.358} C_VEL
LIN {X 0,Y 640.755,Z 411.395,A -85,B 0,C 180,E1 23757.764,E2 23757.764} C_VEL
LIN {X 0,Y 640.795,Z 411.409,A -85,B 0,C 180,E1 23754.628,E2 23754.628} C_VEL
LIN {X 0,Y 640.744,Z 411.401,A -85,B 0,C 180,E1 23751.926,E2 23751.926} C_VEL
LIN {X 0,Y 640.773,Z 411.394,A -85,B 0,C 180,E1 23749.207,E2 23749.207} C_VEL
LIN {X 0,Y 640.755,Z 411.394,A -85,B 0,C 180,E1 23746.003,E2 23746.003} C_VEL
LIN {X 0,Y 640.742,Z 411.401,A -85,B 0,C 180,E1 23743.407,E2 23743.407} C_VEL
LIN {X 0,Y 640.822,Z 411.379,A -85,B 0,C 180,E1 23740.399,E2 23740.399} C_VEL
LIN {X 0,Y 640.74,Z 411.411,A -85,B 0,C 180,E1 23737.425,E2 23737.425} C_VEL
LIN {X 0,Y 640.757,Z 411.388,A -85,B 0,C 180,E1 23734.785,E2 23734.785} C_VEL
LIN {X 0,Y 640.758,Z 411.409,A -85,B 0,C 180,E1 23731.579,E2 23731.579} C_VEL
LIN {X 0,Y 640.733,Z 411.401,A -85,B 0,C 180,E1 23729.004,E2 23729.004} C_VEL
LIN {X 0,Y 640.779,Z 411.389,A -85,B 0,C 180,E1 23726.254,E2 23726.254} C_VEL
LIN {X 0,Y 640.745,Z 411.412,A -85,B 0,C 180,E1 23723.174,E2 23723.174} C_VEL
LIN {X 0,Y 640.763,Z 411.522,A -85,B 0,C 180,E1 23722.4,E2 23722.4} C_VEL
LIN {X 0,Y 642.129,Z 414.921,A -85,B 0,C 180,E1 23721.929,E2 23721.929} C_VEL
LIN {X 0,Y 643.122,Z 416.659,A -85,B 0,C 180,E1 23721.659,E2 23721.659} C_VEL
LIN {X 0,Y 648.594,Z 427.772,A -85,B 0,C 180,E1 23720.11,E2 23720.11} C_VEL
LIN {X 0,Y 662.674,Z 447.78,A -85,B 0,C 180,E1 23718.358,E2 23718.358} C_VEL
LIN {X 0,Y 672.684,Z 462.745,A -85,B 0,C 180,E1 23717.18,E2 23717.18} C_VEL
LIN {X 0,Y 669.197,Z 662.229,A -85,B 0,C 180,E1 23714.484,E2 23714.484} C_VEL
LIN {X 0,Y 665.523,Z 888.106,A -85,B 0,C 180,E1 23711.522,E2 23711.522} C_VEL
LIN {X 0,Y 664.647,Z 918.128,A -85,B 0,C 180,E1 23711.068,E2 23711.068} C_VEL
LIN {X 0,Y 663.609,Z 941.811,A -85,B 0,C 180,E1 23710.572,E2 23710.572} C_VEL
LIN {X 0,Y 662.376,Z 965.246,A -85,B 0,C 180,E1 23709.949,E2 23709.949} C_VEL
LIN {X 0,Y 660.593,Z 993.269,A -85,B 0,C 180,E1 23709.02,E2 23709.02} C_VEL
LIN {X 0,Y 658.9,Z 1016.559,A -85,B 0,C 180,E1 23708.083,E2 23708.083} C_VEL
LIN {X 0,Y 657.243,Z 1037.789,A -85,B 0,C 180,E1 23707.095,E2 23707.095} C_VEL
LIN {X 0,Y 655.286,Z 1061.864,A -85,B 0,C 180,E1 23705.81,E2 23705.81} C_VEL
LIN {X 0,Y 653.158,Z 1085.654,A -85,B 0,C 180,E1 23704.336,E2 23704.336} C_VEL
LIN {X 0,Y 651.429,Z 1104.625,A -85,B 0,C 180,E1 23703.013,E2 23703.013} C_VEL
LIN {X 0,Y 649.713,Z 1123.524,A -85,B 0,C 180,E1 23701.546,E2 23701.546} C_VEL
LIN {X 0,Y 647.703,Z 1146.285,A -85,B 0,C 180,E1 23699.548,E2 23699.548} C_VEL
LIN {X 0,Y 646.288,Z 1162.563,A -85,B 0,C 180,E1 23697.943,E2 23697.943} C_VEL
LIN {X 0,Y 644.954,Z 1178.414,A -85,B 0,C 180,E1 23696.217,E2 23696.217} C_VEL
LIN {X 0,Y 643.597,Z 1196.543,A -85,B 0,C 180,E1 23694.004,E2 23694.004} C_VEL
LIN {X 0,Y 642.552,Z 1211.492,A -85,B 0,C 180,E1 23691.926,E2 23691.926} C_VEL
LIN {X 0,Y 641.766,Z 1224.18,A -85,B 0,C 180,E1 23689.947,E2 23689.947} C_VEL
LIN {X 0,Y 641.052,Z 1237.834,A -85,B 0,C 180,E1 23687.516,E2 23687.516} C_VEL
LIN {X 0,Y 640.591,Z 1248.091,A -85,B 0,C 180,E1 23685.384,E2 23685.384} C_VEL
LIN {X 0,Y 640.295,Z 1256.17,A -85,B 0,C 180,E1 23683.452,E2 23683.452} C_VEL
LIN {X 0,Y 640.138,Z 1263.065,A -85,B 0,C 180,E1 23681.53,E2 23681.53} C_VEL
LIN {X 0,Y 639.97,Z 1269.338,A -85,B 0,C 180,E1 23679.439,E2 23679.439} C_VEL
LIN {X 0,Y 639.951,Z 1274.74,A -85,B 0,C 180,E1 23677.178,E2 23677.178} C_VEL
LIN {X 0,Y 639.915,Z 1278.795,A -85,B 0,C 180,E1 23674.748,E2 23674.748} C_VEL
LIN {X 0,Y 639.909,Z 1280.882,A -85,B 0,C 180,E1 23672.684,E2 23672.684} C_VEL
LIN {X 0,Y 639.868,Z 1281.783,A -85,B 0,C 180,E1 23670.893,E2 23670.893} C_VEL
LIN {X 0,Y 639.868,Z 1281.781,A -85,B 0,C 180,E1 23669.102,E2 23669.102} C_VEL
LIN {X 0,Y 639.909,Z 1280.877,A -85,B 0,C 180,E1 23667.311,E2 23667.311} C_VEL
LIN {X 0,Y 639.914,Z 1278.788,A -85,B 0,C 180,E1 23665.247,E2 23665.247} C_VEL
LIN {X 0,Y 639.951,Z 1274.73,A -85,B 0,C 180,E1 23662.817,E2 23662.817} C_VEL
LIN {X 0,Y 639.969,Z 1269.323,A -85,B 0,C 180,E1 23660.556,E2 23660.556} C_VEL
LIN {X 0,Y 640.128,Z 1263.35,A -85,B 0,C 180,E1 23658.556,E2 23658.556} C_VEL
LIN {X 0,Y 640.292,Z 1256.481,A -85,B 0,C 180,E1 23656.629,E2 23656.629} C_VEL
LIN {X 0,Y 640.578,Z 1248.478,A -85,B 0,C 180,E1 23654.703,E2 23654.703} C_VEL
LIN {X 0,Y 641.011,Z 1238.741,A -85,B 0,C 180,E1 23652.665,E2 23652.665} C_VEL
LIN {X 0,Y 641.712,Z 1225.296,A -85,B 0,C 180,E1 23650.236,E2 23650.236} C_VEL
LIN {X 0,Y 642.509,Z 1212.099,A -85,B 0,C 180,E1 23648.163,E2 23648.163} C_VEL
LIN {X 0,Y 643.486,Z 1197.839,A -85,B 0,C 180,E1 23646.17,E2 23646.17} C_VEL
LIN {X 0,Y 644.817,Z 1180.055,A -85,B 0,C 180,E1 23643.969,E2 23643.969} C_VEL
LIN {X 0,Y 646.221,Z 1163.365,A -85,B 0,C 180,E1 23642.141,E2 23642.141} C_VEL
LIN {X 0,Y 647.71,Z 1146.227,A -85,B 0,C 180,E1 23640.446,E2 23640.446} C_VEL
LIN {X 0,Y 649.719,Z 1123.453,A -85,B 0,C 180,E1 23638.449,E2 23638.449} C_VEL
LIN {X 0,Y 651.436,Z 1104.544,A -85,B 0,C 180,E1 23636.982,E2 23636.982} C_VEL
LIN {X 0,Y 653.164,Z 1085.562,A -85,B 0,C 180,E1 23635.658,E2 23635.658} C_VEL
LIN {X 0,Y 655.293,Z 1061.76,A -85,B 0,C 180,E1 23634.184,E2 23634.184} C_VEL
LIN {X 0,Y 657.18,Z 1038.682,A -85,B 0,C 180,E1 23632.949,E2 23632.949} C_VEL
LIN {X 0,Y 658.828,Z 1017.562,A -85,B 0,C 180,E1 23631.961,E2 23631.961} C_VEL
LIN {X 0,Y 660.418,Z 995.69,A -85,B 0,C 180,E1 23631.073,E2 23631.073} C_VEL
LIN {X 0,Y 662.238,Z 967.997,A -85,B 0,C 180,E1 23630.13,E2 23630.13} C_VEL
LIN {X 0,Y 663.556,Z 942.956,A -85,B 0,C 180,E1 23629.456,E2 23629.456} C_VEL
LIN {X 0,Y 664.581,Z 919.732,A -85,B 0,C 180,E1 23628.962,E2 23628.962} C_VEL
LIN {X 0,Y 665.458,Z 892.216,A -85,B 0,C 180,E1 23628.531,E2 23628.531} C_VEL
LIN {X 0,Y 669.119,Z 666.707,A -85,B 0,C 180,E1 23625.575,E2 23625.575} C_VEL
LIN {X 0,Y 672.582,Z 468.314,A -85,B 0,C 180,E1 23622.896,E2 23622.896} C_VEL
LIN {X 0,Y 672.534,Z 462.382,A -85,B 0,C 180,E1 23622.801,E2 23622.801} C_VEL
LIN {X 0,Y 656.482,Z 438.839,A -85,B 0,C 180,E1 23620.886,E2 23620.886} C_VEL
LIN {X 0,Y 648.021,Z 426.885,A -85,B 0,C 180,E1 23619.788,E2 23619.788} C_VEL
LIN {X 0,Y 643.133,Z 416.635,A -85,B 0,C 180,E1 23618.341,E2 23618.341} C_VEL
LIN {X 0,Y 640.936,Z 412.386,A -85,B 0,C 180,E1 23617.701,E2 23617.701} C_VEL
LIN {X 0,Y 640.738,Z 411.39,A -85,B 0,C 180,E1 23617.556,E2 23617.556} C_VEL
LIN {X 0,Y 640.746,Z 411.398,A -85,B 0,C 180,E1 23614.939,E2 23614.939} C_VEL
LIN {X 0,Y 640.791,Z 411.41,A -85,B 0,C 180,E1 23611.831,E2 23611.831} C_VEL
LIN {X 0,Y 640.747,Z 411.397,A -85,B 0,C 180,E1 23609.087,E2 23609.087} C_VEL
LIN {X 0,Y 640.802,Z 411.389,A -85,B 0,C 180,E1 23606.305,E2 23606.305} C_VEL
LIN {X 0,Y 640.764,Z 411.412,A -85,B 0,C 180,E1 23603.203,E2 23603.203} C_VEL
LIN {X 0,Y 640.769,Z 411.385,A -85,B 0,C 180,E1 23600.555,E2 23600.555} C_VEL
LIN {X 0,Y 640.809,Z 411.406,A -85,B 0,C 180,E1 23597.433,E2 23597.433} C_VEL
LIN {X 0,Y 640.768,Z 411.378,A -85,B 0,C 180,E1 23594.551,E2 23594.551} C_VEL
LIN {X 0,Y 640.831,Z 411.402,A -85,B 0,C 180,E1 23591.517,E2 23591.517} C_VEL
LIN {X 0,Y 640.776,Z 411.379,A -85,B 0,C 180,E1 23588.525,E2 23588.525} C_VEL
LIN {X 0,Y 640.832,Z 411.403,A -85,B 0,C 180,E1 23585.551,E2 23585.551} C_VEL
LIN {X 0,Y 640.785,Z 411.378,A -85,B 0,C 180,E1 23582.504,E2 23582.504} C_VEL
LIN {X 0,Y 640.832,Z 411.405,A -85,B 0,C 180,E1 23579.553,E2 23579.553} C_VEL
LIN {X 0,Y 640.795,Z 411.377,A -85,B 0,C 180,E1 23576.421,E2 23576.421} C_VEL
LIN {X 0,Y 640.827,Z 411.404,A -85,B 0,C 180,E1 23573.37,E2 23573.37} C_VEL
LIN {X 0,Y 640.802,Z 411.378,A -85,B 0,C 180,E1 23570.298,E2 23570.298} C_VEL
LIN {X 0,Y 640.821,Z 411.401,A -85,B 0,C 180,E1 23567.199,E2 23567.199} C_VEL
LIN {X 0,Y 640.811,Z 411.385,A -85,B 0,C 180,E1 23564.153,E2 23564.153} C_VEL
LIN {X 0,Y 640.815,Z 411.394,A -85,B 0,C 180,E1 23561.062,E2 23561.062} C_VEL
LIN {X 0,Y 640.818,Z 411.398,A -85,B 0,C 180,E1 23557.947,E2 23557.947} C_VEL
LIN {X 0,Y 640.807,Z 411.379,A -85,B 0,C 180,E1 23554.886,E2 23554.886} C_VEL
LIN {X 0,Y 640.824,Z 411.407,A -85,B 0,C 180,E1 23551.785,E2 23551.785} C_VEL
LIN {X 0,Y 640.802,Z 411.395,A -85,B 0,C 180,E1 23548.694,E2 23548.694} C_VEL
LIN {X 0,Y 640.824,Z 411.379,A -85,B 0,C 180,E1 23545.609,E2 23545.609} C_VEL
LIN {X 0,Y 640.793,Z 411.387,A -85,B 0,C 180,E1 23542.515,E2 23542.515} C_VEL
LIN {X 0,Y 640.845,Z 411.511,A -85,B 0,C 180,E1 23541.56,E2 23541.56} C_VEL
LIN {X 0,Y 642.026,Z 414.702,A -85,B 0,C 180,E1 23541.124,E2 23541.124} C_VEL
LIN {X 0,Y 643.035,Z 416.392,A -85,B 0,C 180,E1 23540.853,E2 23540.853} C_VEL
LIN {X 0,Y 644.178,Z 418.95,A -85,B 0,C 180,E1 23540.533,E2 23540.533} C_VEL
LIN {X 0,Y 650.561,Z 427.553,A -85,B 0,C 180,E1 23539.708,E2 23539.708} C_VEL
LIN {X 0,Y 661.71,Z 443.14,A -85,B 0,C 180,E1 23538.327,E2 23538.327} C_VEL
LIN {X 0,Y 669.215,Z 454.224,A -85,B 0,C 180,E1 23537.434,E2 23537.434} C_VEL
LIN {X 0,Y 670.12,Z 457.233,A -85,B 0,C 180,E1 23537.303,E2 23537.303} C_VEL
LIN {X 0,Y 669.916,Z 462.288,A -85,B 0,C 180,E1 23537.244,E2 23537.244} C_VEL
LIN {X 0,Y 666.952,Z 475.616,A -85,B 0,C 180,E1 23537.313,E2 23537.313} C_VEL
LIN {X 0,Y 666.765,Z 478.041,A -85,B 0,C 180,E1 23537.292,E2 23537.292} C_VEL
LIN {X 0,Y 662.925,Z 683.193,A -85,B 0,C 180,E1 23534.511,E2 23534.511} C_VEL
LIN {X 0,Y 659.138,Z 892.921,A -85,B 0,C 180,E1 23531.732,E2 23531.732} C_VEL
LIN {X 0,Y 658.207,Z 917.434,A -85,B 0,C 180,E1 23531.305,E2 23531.305} C_VEL
LIN {X 0,Y 656.725,Z 946.103,A -85,B 0,C 180,E1 23530.62,E2 23530.62} C_VEL
LIN {X 0,Y 655.248,Z 969.159,A -85,B 0,C 180,E1 23529.917,E2 23529.917} C_VEL
LIN {X 0,Y 653.792,Z 989.802,A -85,B 0,C 180,E1 23529.171,E2 23529.171} C_VEL
LIN {X 0,Y 652.111,Z 1011.249,A -85,B 0,C 180,E1 23528.274,E2 23528.274} C_VEL
LIN {X 0,Y 649.882,Z 1037.579,A -85,B 0,C 180,E1 23526.984,E2 23526.984} C_VEL
LIN {X 0,Y 647.799,Z 1059.76,A -85,B 0,C 180,E1 23525.719,E2 23525.719} C_VEL
LIN {X 0,Y 646.002,Z 1078.618,A -85,B 0,C 180,E1 23524.508,E2 23524.508} C_VEL
LIN {X 0,Y 644.107,Z 1097.972,A -85,B 0,C 180,E1 23523.124,E2 23523.124} C_VEL
LIN {X 0,Y 641.806,Z 1121.607,A -85,B 0,C 180,E1 23521.206,E2 23521.206} C_VEL
LIN {X 0,Y 640.111,Z 1139.335,A -85,B 0,C 180,E1 23519.579,E2 23519.579} C_VEL
LIN {X 0,Y 638.584,Z 1155.731,A -85,B 0,C 180,E1 23517.917,E2 23517.917} C_VEL
LIN {X 0,Y 636.854,Z 1175.373,A -85,B 0,C 180,E1 23515.681,E2 23515.681} C_VEL
LIN {X 0,Y 635.598,Z 1190.63,A -85,B 0,C 180,E1 23513.712,E2 23513.712} C_VEL
LIN {X 0,Y 634.603,Z 1204.344,A -85,B 0,C 180,E1 23511.734,E2 23511.734} C_VEL
LIN {X 0,Y 633.64,Z 1219.414,A -85,B 0,C 180,E1 23509.259,E2 23509.259} C_VEL
LIN {X 0,Y 633.01,Z 1230.652,A -85,B 0,C 180,E1 23507.128,E2 23507.128} C_VEL
LIN {X 0,Y 632.603,Z 1239.916,A -85,B 0,C 180,E1 23505.119,E2 23505.119} C_VEL
LIN {X 0,Y 632.271,Z 1249.514,A -85,B 0,C 180,E1 23502.7,E2 23502.7} C_VEL
LIN {X 0,Y 632.073,Z 1257.222,A -85,B 0,C 180,E1 23500.276,E2 23500.276} C_VEL
LIN {X 0,Y 631.954,Z 1262.836,A -85,B 0,C 180,E1 23498.097,E2 23498.097} C_VEL
LIN {X 0,Y 631.93,Z 1267.26,A -85,B 0,C 180,E1 23495.814,E2 23495.814} C_VEL
LIN {X 0,Y 631.911,Z 1270.368,A -85,B 0,C 180,E1 23493.359,E2 23493.359} C_VEL
LIN {X 0,Y 631.893,Z 1271.702,A -85,B 0,C 180,E1 23491.181,E2 23491.181} C_VEL
LIN {X 0,Y 631.863,Z 1271.839,A -85,B 0,C 180,E1 23489.277,E2 23489.277} C_VEL
LIN {X 0,Y 631.905,Z 1270.983,A -85,B 0,C 180,E1 23487.373,E2 23487.373} C_VEL
LIN {X 0,Y 631.913,Z 1268.962,A -85,B 0,C 180,E1 23485.283,E2 23485.283} C_VEL
LIN {X 0,Y 631.947,Z 1265.169,A -85,B 0,C 180,E1 23482.914,E2 23482.914} C_VEL
LIN {X 0,Y 631.97,Z 1259.97,A -85,B 0,C 180,E1 23480.624,E2 23480.624} C_VEL
LIN {X 0,Y 632.15,Z 1253.515,A -85,B 0,C 180,E1 23478.415,E2 23478.415} C_VEL
LIN {X 0,Y 632.321,Z 1246.699,A -85,B 0,C 180,E1 23476.469,E2 23476.469} C_VEL
LIN {X 0,Y 632.633,Z 1238.699,A -85,B 0,C 180,E1 23474.511,E2 23474.511} C_VEL
LIN {X 0,Y 633.106,Z 1228.987,A -85,B 0,C 180,E1 23472.447,E2 23472.447} C_VEL
LIN {X 0,Y 633.868,Z 1215.592,A -85,B 0,C 180,E1 23469.986,E2 23469.986} C_VEL
LIN {X 0,Y 634.757,Z 1202.22,A -85,B 0,C 180,E1 23467.856,E2 23467.856} C_VEL
LIN {X 0,Y 635.807,Z 1188.206,A -85,B 0,C 180,E1 23465.869,E2 23465.869} C_VEL
LIN {X 0,Y 637.263,Z 1170.355,A -85,B 0,C 180,E1 23463.628,E2 23463.628} C_VEL
LIN {X 0,Y 638.754,Z 1153.826,A -85,B 0,C 180,E1 23461.792,E2 23461.792} C_VEL
LIN {X 0,Y 640.309,Z 1137.235,A -85,B 0,C 180,E1 23460.127,E2 23460.127} C_VEL
LIN {X 0,Y 642.382,Z 1115.726,A -85,B 0,C 180,E1 23458.198,E2 23458.198} C_VEL
LIN {X 0,Y 644.359,Z 1095.469,A -85,B 0,C 180,E1 23456.6,E2 23456.6} C_VEL
LIN {X 0,Y 646.163,Z 1076.999,A -85,B 0,C 180,E1 23455.293,E2 23455.293} C_VEL
LIN {X 0,Y 648.194,Z 1055.872,A -85,B 0,C 180,E1 23453.955,E2 23453.955} C_VEL
LIN {X 0,Y 650.536,Z 1029.606,A -85,B 0,C 180,E1 23452.513,E2 23452.513} C_VEL
LIN {X 0,Y 652.297,Z 1008.593,A -85,B 0,C 180,E1 23451.518,E2 23451.518} C_VEL
LIN {X 0,Y 653.993,Z 986.855,A -85,B 0,C 180,E1 23450.623,E2 23450.623} C_VEL
LIN {X 0,Y 655.822,Z 961.303,A -85,B 0,C 180,E1 23449.732,E2 23449.732} C_VEL
LIN {X 0,Y 657.361,Z 934.469,A -85,B 0,C 180,E1 23448.99,E2 23448.99} C_VEL
LIN {X 0,Y 658.457,Z 911.367,A -85,B 0,C 180,E1 23448.489,E2 23448.489} C_VEL
LIN {X 0,Y 659.312,Z 887.393,A -85,B 0,C 180,E1 23448.097,E2 23448.097} C_VEL
LIN {X 0,Y 663.275,Z 663.669,A -85,B 0,C 180,E1 23445.137,E2 23445.137} C_VEL
LIN {X 0,Y 667.066,Z 463.178,A -85,B 0,C 180,E1 23442.414,E2 23442.414} C_VEL
LIN {X 0,Y 652.499,Z 441.682,A -85,B 0,C 180,E1 23440.638,E2 23440.638} C_VEL
LIN {X 0,Y 643.809,Z 429.744,A -85,B 0,C 180,E1 23439.522,E2 23439.522} C_VEL
LIN {X 0,Y 635.438,Z 418.248,A -85,B 0,C 180,E1 23438.372,E2 23438.372} C_VEL
LIN {X 0,Y 634.739,Z 416.623,A -85,B 0,C 180,E1 23438.135,E2 23438.135} C_VEL
LIN {X 0,Y 633.142,Z 413.822,A -85,B 0,C 180,E1 23437.674,E2 23437.674} C_VEL
LIN {X 0,Y 632.827,Z 412.399,A -85,B 0,C 180,E1 23437.468,E2 23437.468} C_VEL
LIN {X 0,Y 632.889,Z 412.365,A -85,B 0,C 180,E1 23434.451,E2 23434.451} C_VEL
LIN {X 0,Y 632.828,Z 412.392,A -85,B 0,C 180,E1 23431.427,E2 23431.427} C_VEL
LIN {X 0,Y 632.851,Z 412.388,A -85,B 0,C 180,E1 23428.603,E2 23428.603} C_VEL
LIN {X 0,Y 632.83,Z 412.367,A -85,B 0,C 180,E1 23425.353,E2 23425.353} C_VEL
LIN {X 0,Y 632.833,Z 412.403,A -85,B 0,C 180,E1 23422.578,E2 23422.578} C_VEL
LIN {X 0,Y 632.85,Z 412.377,A -85,B 0,C 180,E1 23419.378,E2 23419.378} C_VEL
LIN {X 0,Y 632.819,Z 412.4,A -85,B 0,C 180,E1 23416.618,E2 23416.618} C_VEL
LIN {X 0,Y 632.894,Z 412.37,A -85,B 0,C 180,E1 23413.615,E2 23413.615} C_VEL
LIN {X 0,Y 632.817,Z 412.395,A -85,B 0,C 180,E1 23410.653,E2 23410.653} C_VEL
LIN {X 0,Y 632.84,Z 412.372,A -85,B 0,C 180,E1 23407.875,E2 23407.875} C_VEL
LIN {X 0,Y 632.829,Z 412.391,A -85,B 0,C 180,E1 23404.713,E2 23404.713} C_VEL
LIN {X 0,Y 632.812,Z 412.374,A -85,B 0,C 180,E1 23401.992,E2 23401.992} C_VEL
LIN {X 0,Y 632.876,Z 412.389,A -85,B 0,C 180,E1 23398.914,E2 23398.914} C_VEL
LIN {X 0,Y 632.805,Z 412.374,A -85,B 0,C 180,E1 23396.013,E2 23396.013} C_VEL
LIN {X 0,Y 632.87,Z 412.397,A -85,B 0,C 180,E1 23393.104,E2 23393.104} C_VEL
LIN {X 0,Y 632.808,Z 412.375,A -85,B 0,C 180,E1 23389.991,E2 23389.991} C_VEL
LIN {X 0,Y 632.818,Z 412.403,A -85,B 0,C 180,E1 23387.313,E2 23387.313} C_VEL
LIN {X 0,Y 632.833,Z 412.373,A -85,B 0,C 180,E1 23384.137,E2 23384.137} C_VEL
LIN {X 0,Y 632.803,Z 412.4,A -85,B 0,C 180,E1 23381.387,E2 23381.387} C_VEL
LIN {X 0,Y 632.887,Z 412.369,A -85,B 0,C 180,E1 23378.401,E2 23378.401} C_VEL
LIN {X 0,Y 632.802,Z 412.387,A -85,B 0,C 180,E1 23375.445,E2 23375.445} C_VEL
LIN {X 0,Y 632.817,Z 412.397,A -85,B 0,C 180,E1 23372.728,E2 23372.728} C_VEL
LIN {X 0,Y 632.809,Z 412.379,A -85,B 0,C 180,E1 23369.435,E2 23369.435} C_VEL
LIN {X 0,Y 632.797,Z 412.392,A -85,B 0,C 180,E1 23366.858,E2 23366.858} C_VEL
LIN {X 0,Y 632.878,Z 412.399,A -85,B 0,C 180,E1 23363.828,E2 23363.828} C_VEL
LIN {X 0,Y 632.839,Z 412.61,A -85,B 0,C 180,E1 23363.224,E2 23363.224} C_VEL
LIN {X 0,Y 634.182,Z 416.005,A -85,B 0,C 180,E1 23362.739,E2 23362.739} C_VEL
LIN {X 0,Y 635.183,Z 417.641,A -85,B 0,C 180,E1 23362.468,E2 23362.468} C_VEL
LIN {X 0,Y 637.591,Z 422.661,A -85,B 0,C 180,E1 23361.724,E2 23361.724} C_VEL
LIN {X 0,Y 640.093,Z 427.7,A -85,B 0,C 180,E1 23361.028,E2 23361.028} C_VEL
LIN {X 0,Y 649.761,Z 441.078,A -85,B 0,C 180,E1 23359.764,E2 23359.764} C_VEL
LIN {X 0,Y 663.396,Z 460.848,A -85,B 0,C 180,E1 23358.081,E2 23358.081} C_VEL
LIN {X 0,Y 667.156,Z 466.737,A -85,B 0,C 180,E1 23357.631,E2 23357.631} C_VEL
LIN {X 0,Y 663.436,Z 664.936,A -85,B 0,C 180,E1 23354.935,E2 23354.935} C_VEL
LIN {X 0,Y 659.492,Z 890.523,A -85,B 0,C 180,E1 23351.953,E2 23351.953} C_VEL
LIN {X 0,Y 658.56,Z 918.98,A -85,B 0,C 180,E1 23351.511,E2 23351.511} C_VEL
LIN {X 0,Y 657.471,Z 942.211,A -85,B 0,C 180,E1 23351.019,E2 23351.019} C_VEL
LIN {X 0,Y 656.162,Z 965.468,A -85,B 0,C 180,E1 23350.397,E2 23350.397} C_VEL
LIN {X 0,Y 654.277,Z 993.266,A -85,B 0,C 180,E1 23349.47,E2 23349.47} C_VEL
LIN {X 0,Y 652.461,Z 1016.556,A -85,B 0,C 180,E1 23348.527,E2 23348.527} C_VEL
LIN {X 0,Y 650.697,Z 1037.615,A -85,B 0,C 180,E1 23347.541,E2 23347.541} C_VEL
LIN {X 0,Y 648.61,Z 1061.356,A -85,B 0,C 180,E1 23346.268,E2 23346.268} C_VEL
LIN {X 0,Y 646.313,Z 1085.469,A -85,B 0,C 180,E1 23344.765,E2 23344.765} C_VEL
LIN {X 0,Y 644.511,Z 1103.956,A -85,B 0,C 180,E1 23343.466,E2 23343.466} C_VEL
LIN {X 0,Y 642.772,Z 1121.709,A -85,B 0,C 180,E1 23342.084,E2 23342.084} C_VEL
LIN {X 0,Y 640.754,Z 1142.726,A -85,B 0,C 180,E1 23340.263,E2 23340.263} C_VEL
LIN {X 0,Y 638.913,Z 1162.027,A -85,B 0,C 180,E1 23338.353,E2 23338.353} C_VEL
LIN {X 0,Y 637.496,Z 1177.839,A -85,B 0,C 180,E1 23336.616,E2 23336.616} C_VEL
LIN {X 0,Y 636.018,Z 1195.751,A -85,B 0,C 180,E1 23334.419,E2 23334.419} C_VEL
LIN {X 0,Y 634.854,Z 1210.85,A -85,B 0,C 180,E1 23332.303,E2 23332.303} C_VEL
LIN {X 0,Y 633.98,Z 1223.604,A -85,B 0,C 180,E1 23330.299,E2 23330.299} C_VEL
LIN {X 0,Y 633.203,Z 1236.905,A -85,B 0,C 180,E1 23327.931,E2 23327.931} C_VEL
LIN {X 0,Y 632.663,Z 1248.092,A -85,B 0,C 180,E1 23325.582,E2 23325.582} C_VEL
LIN {X 0,Y 632.33,Z 1256.171,A -85,B 0,C 180,E1 23323.624,E2 23323.624} C_VEL
LIN {X 0,Y 632.161,Z 1263.064,A -85,B 0,C 180,E1 23321.677,E2 23321.677} C_VEL
LIN {X 0,Y 631.984,Z 1269.337,A -85,B 0,C 180,E1 23319.559,E2 23319.559} C_VEL
LIN {X 0,Y 631.947,Z 1274.74,A -85,B 0,C 180,E1 23317.269,E2 23317.269} C_VEL
LIN {X 0,Y 631.916,Z 1278.792,A -85,B 0,C 180,E1 23314.808,E2 23314.808} C_VEL
LIN {X 0,Y 631.909,Z 1280.882,A -85,B 0,C 180,E1 23312.718,E2 23312.718} C_VEL
LIN {X 0,Y 631.868,Z 1281.783,A -85,B 0,C 180,E1 23310.904,E2 23310.904} C_VEL
LIN {X 0,Y 631.869,Z 1281.781,A -85,B 0,C 180,E1 23309.091,E2 23309.091} C_VEL
LIN {X 0,Y 631.909,Z 1280.878,A -85,B 0,C 180,E1 23307.277,E2 23307.277} C_VEL
LIN {X 0,Y 631.916,Z 1278.785,A -85,B 0,C 180,E1 23305.187,E2 23305.187} C_VEL
LIN {X 0,Y 631.948,Z 1274.73,A -85,B 0,C 180,E1 23302.726,E2 23302.726} C_VEL
LIN {X 0,Y 631.986,Z 1269.323,A -85,B 0,C 180,E1 23300.435,E2 23300.435} C_VEL
LIN {X 0,Y 632.161,Z 1263.046,A -85,B 0,C 180,E1 23298.317,E2 23298.317} C_VEL
LIN {X 0,Y 632.33,Z 1256.149,A -85,B 0,C 180,E1 23296.37,E2 23296.37} C_VEL
LIN {X 0,Y 632.664,Z 1248.069,A -85,B 0,C 180,E1 23294.413,E2 23294.413} C_VEL
LIN {X 0,Y 633.204,Z 1236.881,A -85,B 0,C 180,E1 23292.064,E2 23292.064} C_VEL
LIN {X 0,Y 633.95,Z 1224.148,A -85,B 0,C 180,E1 23289.791,E2 23289.791} C_VEL
LIN {X 0,Y 634.812,Z 1211.458,A -85,B 0,C 180,E1 23287.787,E2 23287.787} C_VEL
LIN {X 0,Y 635.963,Z 1196.42,A -85,B 0,C 180,E1 23285.672,E2 23285.672} C_VEL
LIN {X 0,Y 637.445,Z 1178.363,A -85,B 0,C 180,E1 23283.444,E2 23283.444} C_VEL
LIN {X 0,Y 638.877,Z 1162.438,A -85,B 0,C 180,E1 23281.69,E2 23281.69} C_VEL
LIN {X 0,Y 640.696,Z 1143.246,A -85,B 0,C 180,E1 23279.787,E2 23279.787} C_VEL
LIN {X 0,Y 642.717,Z 1122.244,A -85,B 0,C 180,E1 23277.959,E2 23277.959} C_VEL
LIN {X 0,Y 644.452,Z 1104.541,A -85,B 0,C 180,E1 23276.577,E2 23276.577} C_VEL
LIN {X 0,Y 646.231,Z 1086.294,A -85,B 0,C 180,E1 23275.291,E2 23275.291} C_VEL
LIN {X 0,Y 648.435,Z 1063.485,A -85,B 0,C 180,E1 23273.855,E2 23273.855} C_VEL
LIN {X 0,Y 650.613,Z 1038.679,A -85,B 0,C 180,E1 23272.511,E2 23272.511} C_VEL
LIN {X 0,Y 652.38,Z 1017.559,A -85,B 0,C 180,E1 23271.517,E2 23271.517} C_VEL
LIN {X 0,Y 654.081,Z 995.686,A -85,B 0,C 180,E1 23270.623,E2 23270.623} C_VEL
LIN {X 0,Y 656.022,Z 968.145,A -85,B 0,C 180,E1 23269.681,E2 23269.681} C_VEL
LIN {X 0,Y 657.416,Z 943.328,A -85,B 0,C 180,E1 23269.007,E2 23269.007} C_VEL
LIN {X 0,Y 658.501,Z 920.357,A -85,B 0,C 180,E1 23268.515,E2 23268.515} C_VEL
LIN {X 0,Y 659.413,Z 894.219,A -85,B 0,C 180,E1 23268.096,E2 23268.096} C_VEL
LIN {X 0,Y 663.367,Z 668.648,A -85,B 0,C 180,E1 23265.115,E2 23265.115} C_VEL
LIN {X 0,Y 667.072,Z 471.04,A -85,B 0,C 180,E1 23262.428,E2 23262.428} C_VEL
LIN {X 0,Y 667.06,Z 466.279,A -85,B 0,C 180,E1 23262.353,E2 23262.353} C_VEL
LIN {X 0,Y 651.905,Z 444.157,A -85,B 0,C 180,E1 23260.509,E2 23260.509} C_VEL
LIN {X 0,Y 641.981,Z 430.246,A -85,B 0,C 180,E1 23259.224,E2 23259.224} C_VEL
LIN {X 0,Y 639.582,Z 426.739,A -85,B 0,C 180,E1 23258.872,E2 23258.872} C_VEL
LIN {X 0,Y 636.478,Z 420.412,A -85,B 0,C 180,E1 23257.942,E2 23257.942} C_VEL
LIN {X 0,Y 634.55,Z 416.469,A -85,B 0,C 180,E1 23257.349,E2 23257.349} C_VEL
LIN {X 0,Y 633.031,Z 413.496,A -85,B 0,C 180,E1 23256.886,E2 23256.886} C_VEL
LIN {X 0,Y 632.824,Z 412.387,A -85,B 0,C 180,E1 23256.751,E2 23256.751} C_VEL
LIN {X 0,Y 632.814,Z 412.379,A -85,B 0,C 180,E1 23253.575,E2 23253.575} C_VEL
LIN {X 0,Y 632.811,Z 412.387,A -85,B 0,C 180,E1 23250.899,E2 23250.899} C_VEL
LIN {X 0,Y 632.88,Z 412.4,A -85,B 0,C 180,E1 23247.882,E2 23247.882} C_VEL
LIN {X 0,Y 632.814,Z 412.372,A -85,B 0,C 180,E1 23244.911,E2 23244.911} C_VEL
LIN {X 0,Y 632.898,Z 412.383,A -85,B 0,C 180,E1 23241.891,E2 23241.891} C_VEL
LIN {X 0,Y 632.825,Z 412.391,A -85,B 0,C 180,E1 23238.837,E2 23238.837} C_VEL
LIN {X 0,Y 632.891,Z 412.368,A -85,B 0,C 180,E1 23235.862,E2 23235.862} C_VEL
LIN {X 0,Y 632.837,Z 412.395,A -85,B 0,C 180,E1 23232.78,E2 23232.78} C_VEL
LIN {X 0,Y 632.884,Z 412.364,A -85,B 0,C 180,E1 23229.824,E2 23229.824} C_VEL
LIN {X 0,Y 632.848,Z 412.395,A -85,B 0,C 180,E1 23226.714,E2 23226.714} C_VEL
LIN {X 0,Y 632.884,Z 412.363,A -85,B 0,C 180,E1 23223.714,E2 23223.714} C_VEL
LIN {X 0,Y 632.854,Z 412.394,A -85,B 0,C 180,E1 23220.543,E2 23220.543} C_VEL
LIN {X 0,Y 632.885,Z 412.362,A -85,B 0,C 180,E1 23217.555,E2 23217.555} C_VEL
LIN {X 0,Y 632.861,Z 412.394,A -85,B 0,C 180,E1 23214.378,E2 23214.378} C_VEL
LIN {X 0,Y 632.884,Z 412.361,A -85,B 0,C 180,E1 23211.368,E2 23211.368} C_VEL
LIN {X 0,Y 632.87,Z 412.394,A -85,B 0,C 180,E1 23208.24,E2 23208.24} C_VEL
LIN {X 0,Y 632.877,Z 412.363,A -85,B 0,C 180,E1 23205.17,E2 23205.17} C_VEL
LIN {X 0,Y 632.874,Z 412.396,A -85,B 0,C 180,E1 23202.01,E2 23202.01} C_VEL
LIN {X 0,Y 632.873,Z 412.369,A -85,B 0,C 180,E1 23198.983,E2 23198.983} C_VEL
LIN {X 0,Y 632.882,Z 412.389,A -85,B 0,C 180,E1 23195.945,E2 23195.945} C_VEL
LIN {X 0,Y 632.869,Z 412.392,A -85,B 0,C 180,E1 23192.811,E2 23192.811} C_VEL
LIN {X 0,Y 632.883,Z 412.365,A -85,B 0,C 180,E1 23189.736,E2 23189.736} C_VEL
LIN {X 0,Y 632.861,Z 412.382,A -85,B 0,C 180,E1 23186.645,E2 23186.645} C_VEL
LIN {X 0,Y 632.889,Z 412.397,A -85,B 0,C 180,E1 23183.53,E2 23183.53} C_VEL
LIN {X 0,Y 632.874,Z 412.534,A -85,B 0,C 180,E1 23182.393,E2 23182.393} C_VEL
LIN {X 0,Y 634.101,Z 415.738,A -85,B 0,C 180,E1 23181.935,E2 23181.935} C_VEL
LIN {X 0,Y 635.236,Z 417.659,A -85,B 0,C 180,E1 23181.617,E2 23181.617} C_VEL
LIN {X 0,Y 636.259,Z 419.642,A -85,B 0,C 180,E1 23181.399,E2 23181.399} C_VEL
LIN {X 0,Y 646.764,Z 433.756,A -85,B 0,C 180,E1 23180.003,E2 23180.003} C_VEL
LIN {X 0,Y 658.777,Z 450.738,A -85,B 0,C 180,E1 23178.493,E2 23178.493} C_VEL
LIN {X 0,Y 667.061,Z 463.453,A -85,B 0,C 180,E1 23177.493,E2 23177.493} C_VEL
LIN {X 0,Y 666.765,Z 478.041,A -85,B 0,C 180,E1 23177.292,E2 23177.292} C_VEL
LIN {X 0,Y 665.93,Z 485.748,A -85,B 0,C 180,E1 23177.25,E2 23177.25} C_VEL
LIN {X 0,Y 661.265,Z 506.436,A -85,B 0,C 180,E1 23177.365,E2 23177.365} C_VEL
LIN {X 0,Y 660.624,Z 513.045,A -85,B 0,C 180,E1 23177.321,E2 23177.321} C_VEL
LIN {X 0,Y 656.386,Z 726.814,A -85,B 0,C 180,E1 23174.417,E2 23174.417} C_VEL
LIN {X 0,Y 653.115,Z 894.614,A -85,B 0,C 180,E1 23172.176,E2 23172.176} C_VEL
LIN {X 0,Y 652.029,Z 921.37,A -85,B 0,C 180,E1 23171.692,E2 23171.692} C_VEL
LIN {X 0,Y 650.477,Z 947.952,A -85,B 0,C 180,E1 23171.032,E2 23171.032} C_VEL
LIN {X 0,Y 648.982,Z 969.915,A -85,B 0,C 180,E1 23170.353,E2 23170.353} C_VEL
LIN {X 0,Y 647.471,Z 989.815,A -85,B 0,C 180,E1 23169.629,E2 23169.629} C_VEL
LIN {X 0,Y 645.616,Z 1012.108,A -85,B 0,C 180,E1 23168.687,E2 23168.687} C_VEL
LIN {X 0,Y 643.212,Z 1038.486,A -85,B 0,C 180,E1 23167.377,E2 23167.377} C_VEL
LIN {X 0,Y 641.135,Z 1059.312,A -85,B 0,C 180,E1 23166.179,E2 23166.179} C_VEL
LIN {X 0,Y 639.227,Z 1077.964,A -85,B 0,C 180,E1 23164.975,E2 23164.975} C_VEL
LIN {X 0,Y 637.275,Z 1096.653,A -85,B 0,C 180,E1 23163.633,E2 23163.633} C_VEL
LIN {X 0,Y 635.012,Z 1118.29,A -85,B 0,C 180,E1 23161.896,E2 23161.896} C_VEL
LIN {X 0,Y 632.916,Z 1138.327,A -85,B 0,C 180,E1 23160.054,E2 23160.054} C_VEL
LIN {X 0,Y 631.3,Z 1154.347,A -85,B 0,C 180,E1 23158.423,E2 23158.423} C_VEL
LIN {X 0,Y 629.579,Z 1172.288,A -85,B 0,C 180,E1 23156.396,E2 23156.396} C_VEL
LIN {X 0,Y 628.038,Z 1189.655,A -85,B 0,C 180,E1 23154.154,E2 23154.154} C_VEL
LIN {X 0,Y 626.96,Z 1203.076,A -85,B 0,C 180,E1 23152.21,E2 23152.21} C_VEL
LIN {X 0,Y 625.957,Z 1217.319,A -85,B 0,C 180,E1 23149.893,E2 23149.893} C_VEL
LIN {X 0,Y 625.168,Z 1229.923,A -85,B 0,C 180,E1 23147.501,E2 23147.501} C_VEL
